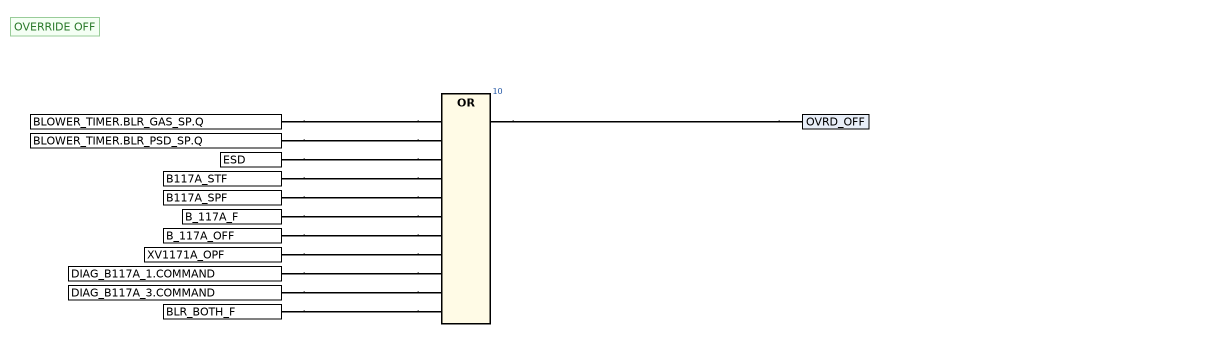
// AUTO ON
(* (BST_S_01.COMMAND OR BST_P_01.COMMAND) AND B117A_SEL OR (BST_S_01.COMPLETE OR BST_P_01.COMPLETE) AND B117A_SEL AND (B117B_STF OR XV1171B_OPF OR B_117B_OFF OR B_117B_F); result not used *)
// AUTO OFF
(* (BSP_S_10.COMMAND OR BSP_P_10.COMMAND) AND XV1171A_CLD; result not used *)
// OVERRIDE ON
(* BLOWER_TIMER.BLR_GAS_SET.Q1 AND B117A_SEL OR DIAG_B117A_2.COMMAND; result not used *)
// OVERRIDE OFF
(* BLOWER_TIMER.BLR_GAS_SP.Q OR BLOWER_TIMER.BLR_PSD_SP.Q OR ESD OR B117A_STF OR B117A_SPF OR B_117A_F OR B_117A_OFF OR XV1171A_OPF OR DIAG_B117A_1.COMMAND OR DIAG_B117A_3.COMMAND OR BLR_BOTH_F; result not used *)
B117A(
    FULL_AUTO := FULL_AUTO,
    SET_AUTO := MP_B117A_A,
    SET_MANUAL := MP_B117A_M,
    AUTO_ON := _w1,
    MANUAL_ON := MP_B117A_ST,
    INHIBIT_ON := MAINTENANCE,
    OVERRIDE_ON := _w2,
    AUTO_OFF := _w3,
    MANUAL_OFF := MP_B117A_SP,
    INHIBIT_OFF := MAINTENANCE,
    OVERRIDE_OFF := _w4,
    FEEDBACK_ON := B_117A_RUN,
    FEEDBACK_OFF := NOT B_117A_RUN); // BWTS.DEVICE
B_117A_ST := B117A.COMMAND_ON;
B117A_A := B117A.AUTO_MODE;
B117A_M := B117A.MANUAL_MODE;
B117A_RUN := B117A.INDICATOR_ON;
B117A_SPD := B117A.INDICATOR_OFF;

END_PROGRAM

// Device/Application/Logic/0.ETC/BLOWER_TIMER
PROGRAM BLOWER_TIMER
VAR
	BLR_GAS_SP: TON;
	BLR_GAS_SET: RS;		// GAS OPERATING ON
	SR_0: SR;
	BLR_PSD_SP: TON;
END_VAR
VAR // added by the converter: edge detectors and wires of the graphical bodies
    _w1 : BOOL;
END_VAR

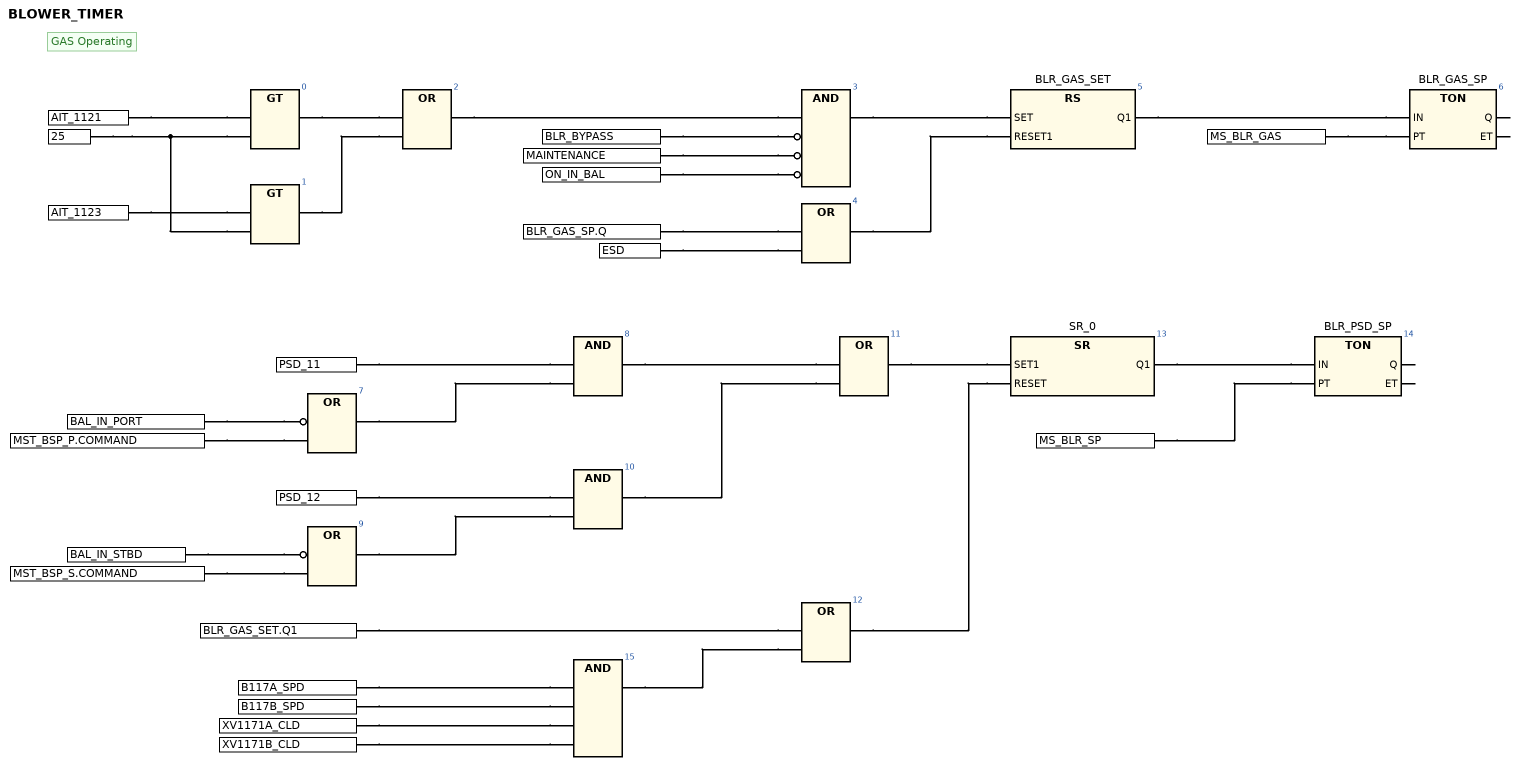
// GAS Operating
BLR_GAS_SET(SET := (AIT_1121 > 25 OR AIT_1123 > 25) AND NOT BLR_BYPASS AND NOT MAINTENANCE AND NOT ON_IN_BAL, RESET1 := BLR_GAS_SP.Q OR ESD); // RS
BLR_GAS_SP(IN := BLR_GAS_SET.Q1, PT := MS_BLR_GAS); // TON
SR_0(SET1 := PSD_11 AND (NOT BAL_IN_PORT OR MST_BSP_P.COMMAND) OR PSD_12 AND (NOT BAL_IN_STBD OR MST_BSP_S.COMMAND), RESET := BLR_GAS_SET.Q1 OR _w1); // SR
BLR_PSD_SP(IN := SR_0.Q1, PT := MS_BLR_SP); // TON
_w1 := B117A_SPD AND B117B_SPD AND XV1171A_CLD AND XV1171B_CLD;

END_PROGRAM

// Device/Application/Logic/4.Device/DEVICE_B117B
PROGRAM DEVICE_B117B
VAR
	B117B : BWTS.DEVICE;
END_VAR
VAR // added by the converter: edge detectors and wires of the graphical bodies
    _w1, _w2, _w3, _w4 : ANY;
END_VAR

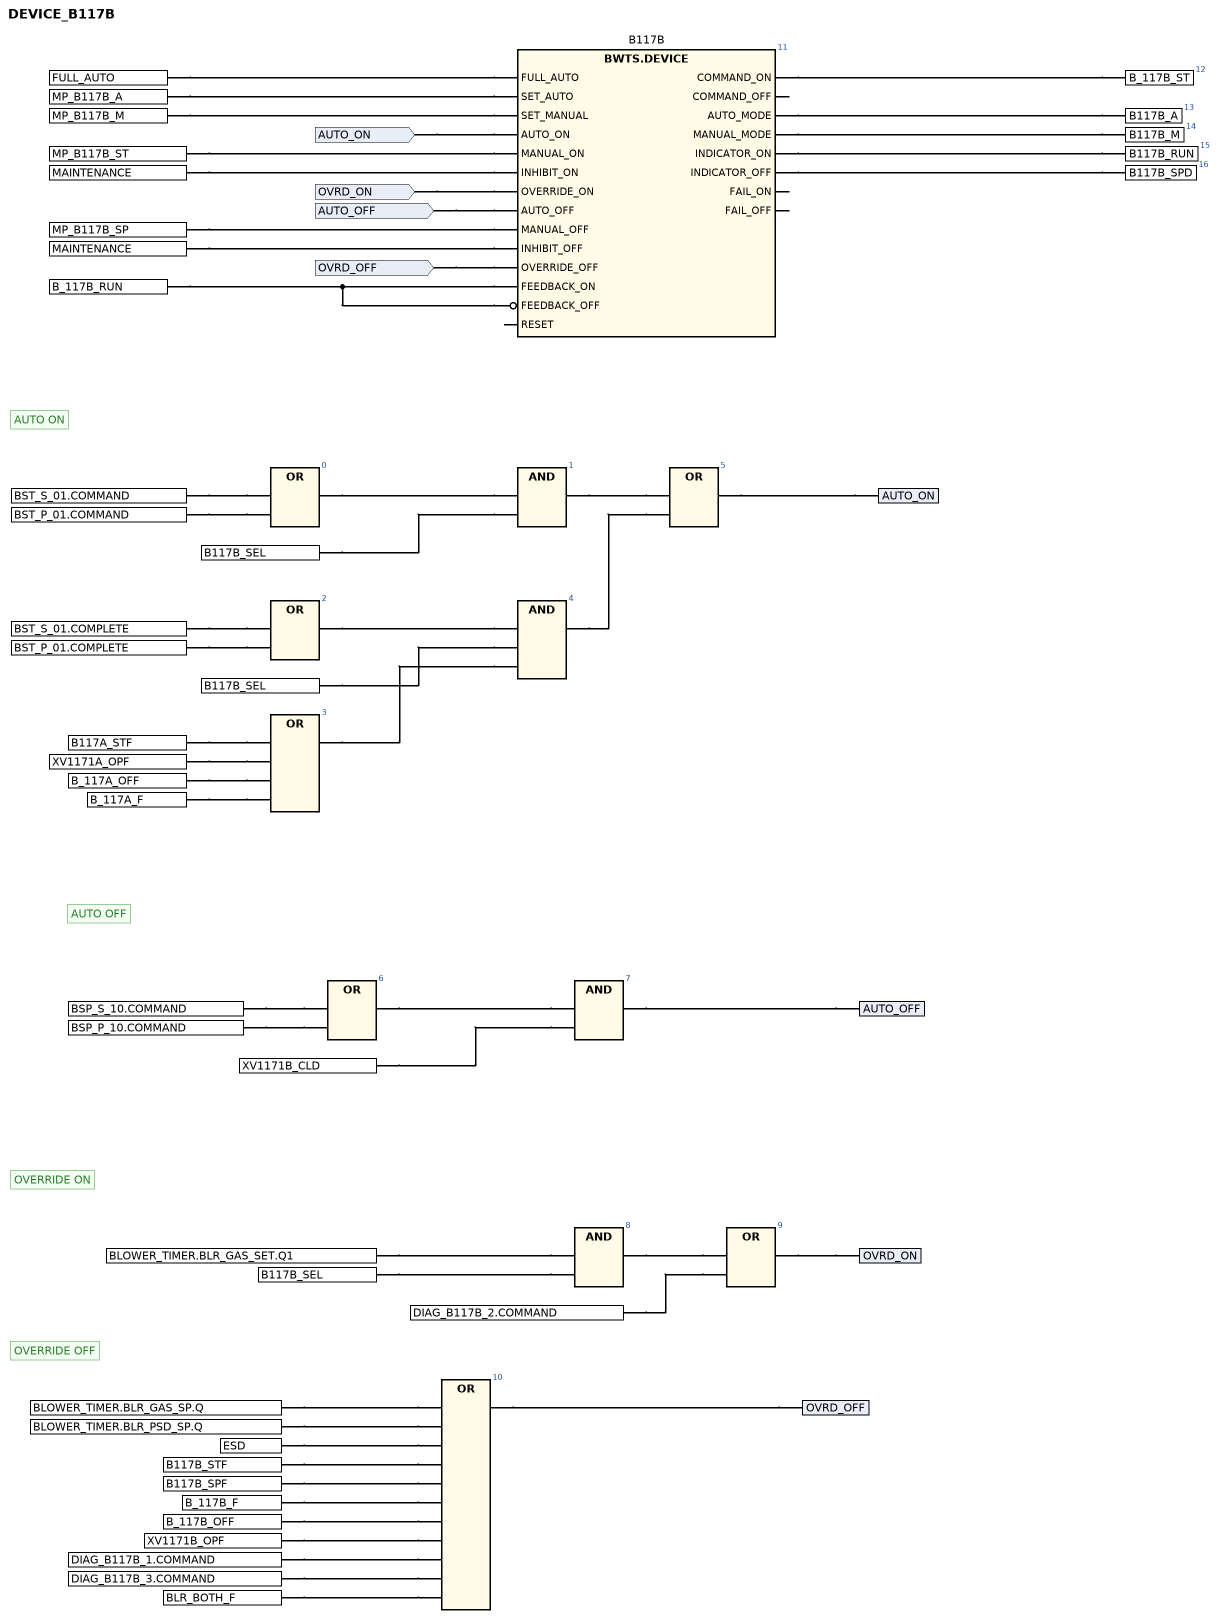
// AUTO ON
(* (BST_S_01.COMMAND OR BST_P_01.COMMAND) AND B117B_SEL OR (BST_S_01.COMPLETE OR BST_P_01.COMPLETE) AND B117B_SEL AND (B117A_STF OR XV1171A_OPF OR B_117A_OFF OR B_117A_F); result not used *)
// AUTO OFF
(* (BSP_S_10.COMMAND OR BSP_P_10.COMMAND) AND XV1171B_CLD; result not used *)
// OVERRIDE ON
(* BLOWER_TIMER.BLR_GAS_SET.Q1 AND B117B_SEL OR DIAG_B117B_2.COMMAND; result not used *)
// OVERRIDE OFF
(* BLOWER_TIMER.BLR_GAS_SP.Q OR BLOWER_TIMER.BLR_PSD_SP.Q OR ESD OR B117B_STF OR B117B_SPF OR B_117B_F OR B_117B_OFF OR XV1171B_OPF OR DIAG_B117B_1.COMMAND OR DIAG_B117B_3.COMMAND OR BLR_BOTH_F; result not used *)
B117B(
    FULL_AUTO := FULL_AUTO,
    SET_AUTO := MP_B117B_A,
    SET_MANUAL := MP_B117B_M,
    AUTO_ON := _w1,
    MANUAL_ON := MP_B117B_ST,
    INHIBIT_ON := MAINTENANCE,
    OVERRIDE_ON := _w2,
    AUTO_OFF := _w3,
    MANUAL_OFF := MP_B117B_SP,
    INHIBIT_OFF := MAINTENANCE,
    OVERRIDE_OFF := _w4,
    FEEDBACK_ON := B_117B_RUN,
    FEEDBACK_OFF := NOT B_117B_RUN); // BWTS.DEVICE
B_117B_ST := B117B.COMMAND_ON;
B117B_A := B117B.AUTO_MODE;
B117B_M := B117B.MANUAL_MODE;
B117B_RUN := B117B.INDICATOR_ON;
B117B_SPD := B117B.INDICATOR_OFF;

END_PROGRAM

// Device/Application/Logic/4.Device/DEVICE_P171A
PROGRAM DEVICE_P171A
VAR
	P171A: BWTS.DEVICE;	
	TON_0: TON;
END_VAR
VAR // added by the converter: edge detectors and wires of the graphical bodies
    _w1, _w2, _w3, _w4, _w5 : BOOL;
    _w6, _w7, _w8, _w9 : ANY;
END_VAR

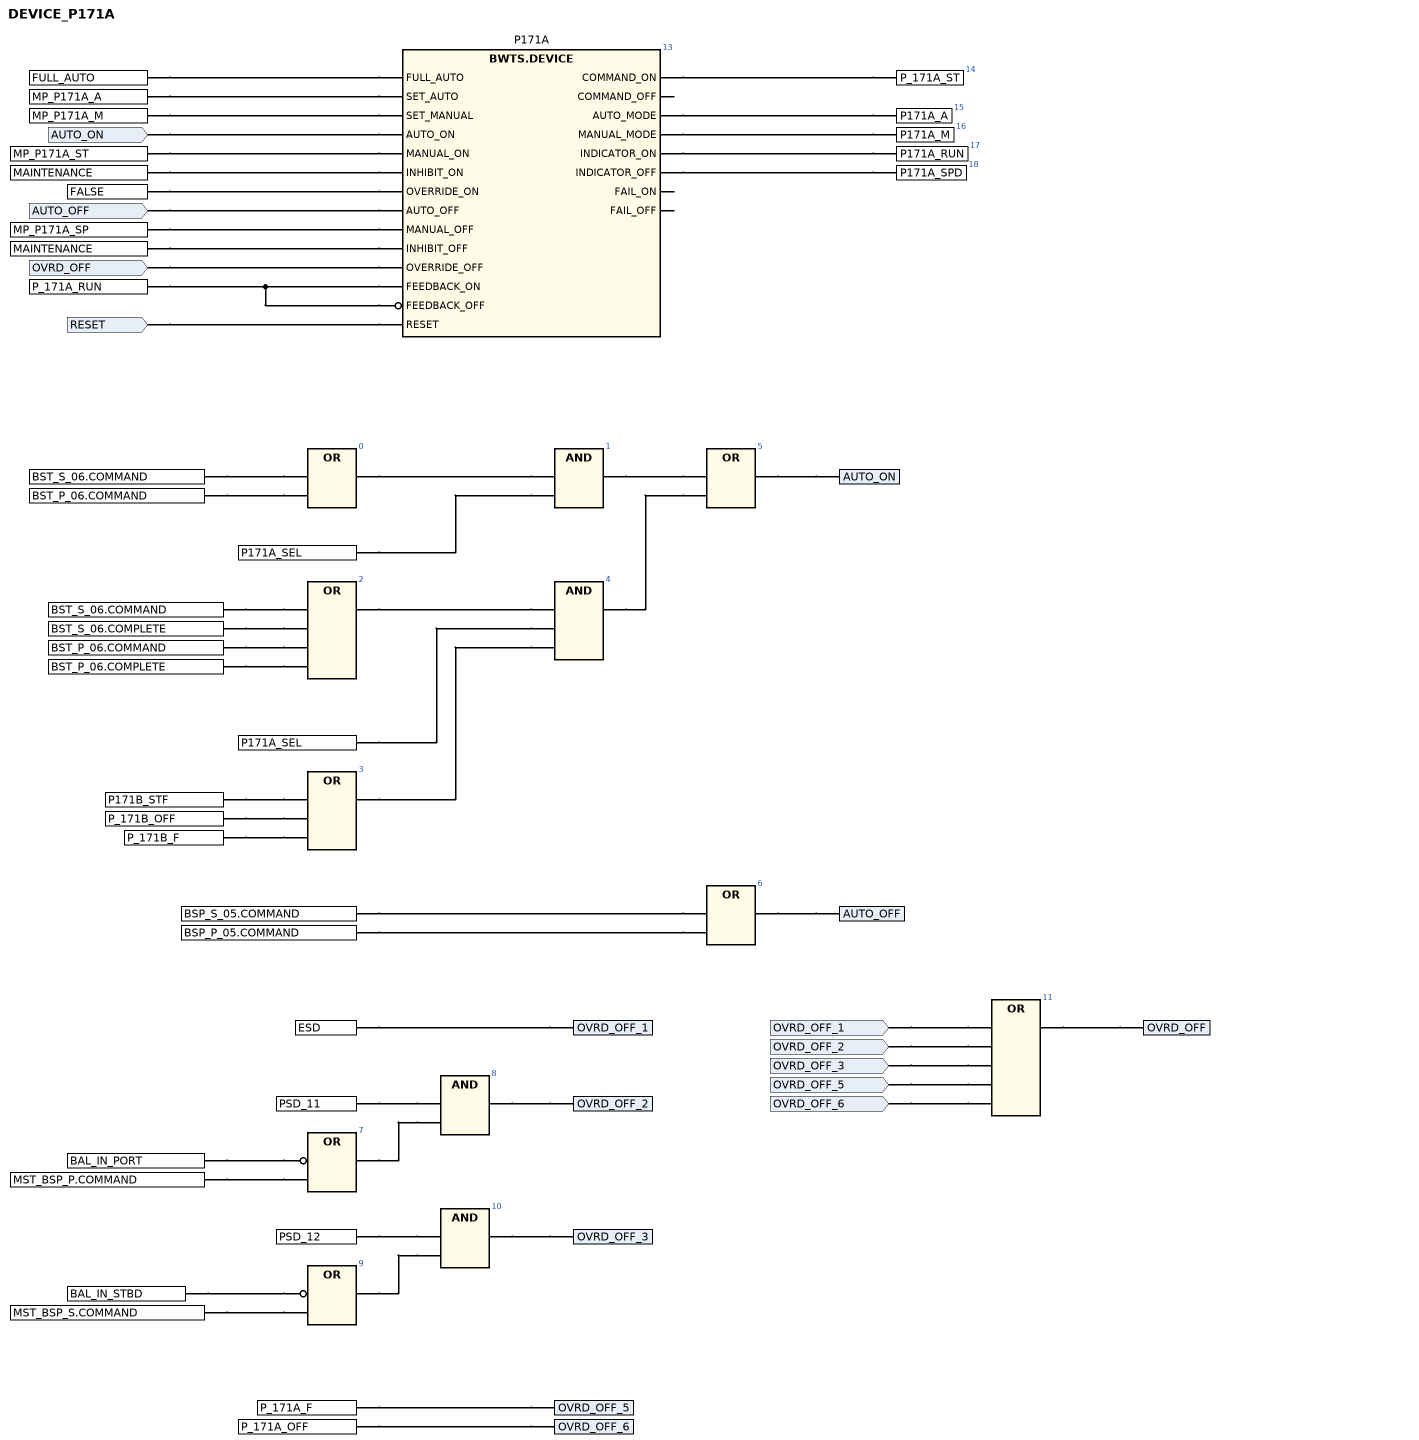
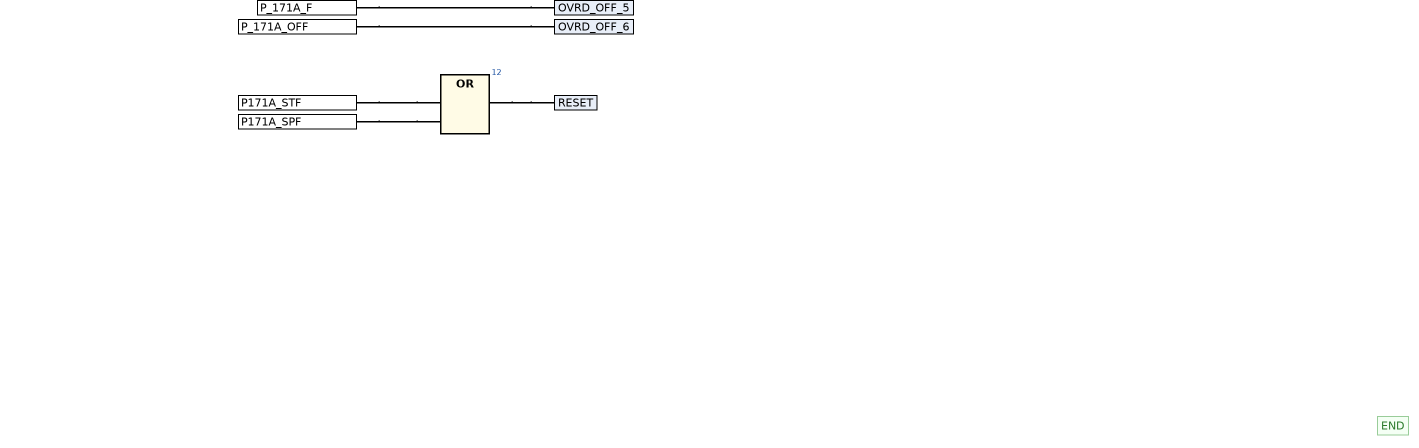
(* (BST_S_06.COMMAND OR BST_P_06.COMMAND) AND P171A_SEL OR (BST_S_06.COMMAND OR BST_S_06.COMPLETE OR BST_P_06.COMMAND OR BST_P_06.COMPLETE) AND P171A_SEL AND (P171B_STF OR P_171B_OFF OR P_171B_F); result not used *)
(* BSP_S_05.COMMAND OR BSP_P_05.COMMAND; result not used *)
(* PSD_11 AND (NOT BAL_IN_PORT OR MST_BSP_P.COMMAND); result not used *)
(* PSD_12 AND (NOT BAL_IN_STBD OR MST_BSP_S.COMMAND); result not used *)
(* _w1 OR _w2 OR _w3 OR _w4 OR _w5; result not used *)
// END
(* P171A_STF OR P171A_SPF; result not used *)
P171A(
    FULL_AUTO := FULL_AUTO,
    SET_AUTO := MP_P171A_A,
    SET_MANUAL := MP_P171A_M,
    AUTO_ON := _w6,
    MANUAL_ON := MP_P171A_ST,
    INHIBIT_ON := MAINTENANCE,
    OVERRIDE_ON := FALSE,
    AUTO_OFF := _w7,
    MANUAL_OFF := MP_P171A_SP,
    INHIBIT_OFF := MAINTENANCE,
    OVERRIDE_OFF := _w8,
    FEEDBACK_ON := P_171A_RUN,
    FEEDBACK_OFF := NOT P_171A_RUN,
    RESET := _w9); // BWTS.DEVICE
P_171A_ST := P171A.COMMAND_ON;
P171A_A := P171A.AUTO_MODE;
P171A_M := P171A.MANUAL_MODE;
P171A_RUN := P171A.INDICATOR_ON;
P171A_SPD := P171A.INDICATOR_OFF;

END_PROGRAM

// Device/Application/Logic/4.Device/DEVICE_P171B
PROGRAM DEVICE_P171B
VAR
	P171B : BWTS.DEVICE;
	AUTO_ON : BOOL;
	AUTO_OFF : BOOL;
	OVRD_OFF : BOOL;
	
	
END_VAR
VAR // added by the converter: edge detectors and wires of the graphical bodies
    _w1, _w2, _w3, _w4, _w5 : BOOL;
    _w6, _w7, _w8, _w9 : ANY;
END_VAR

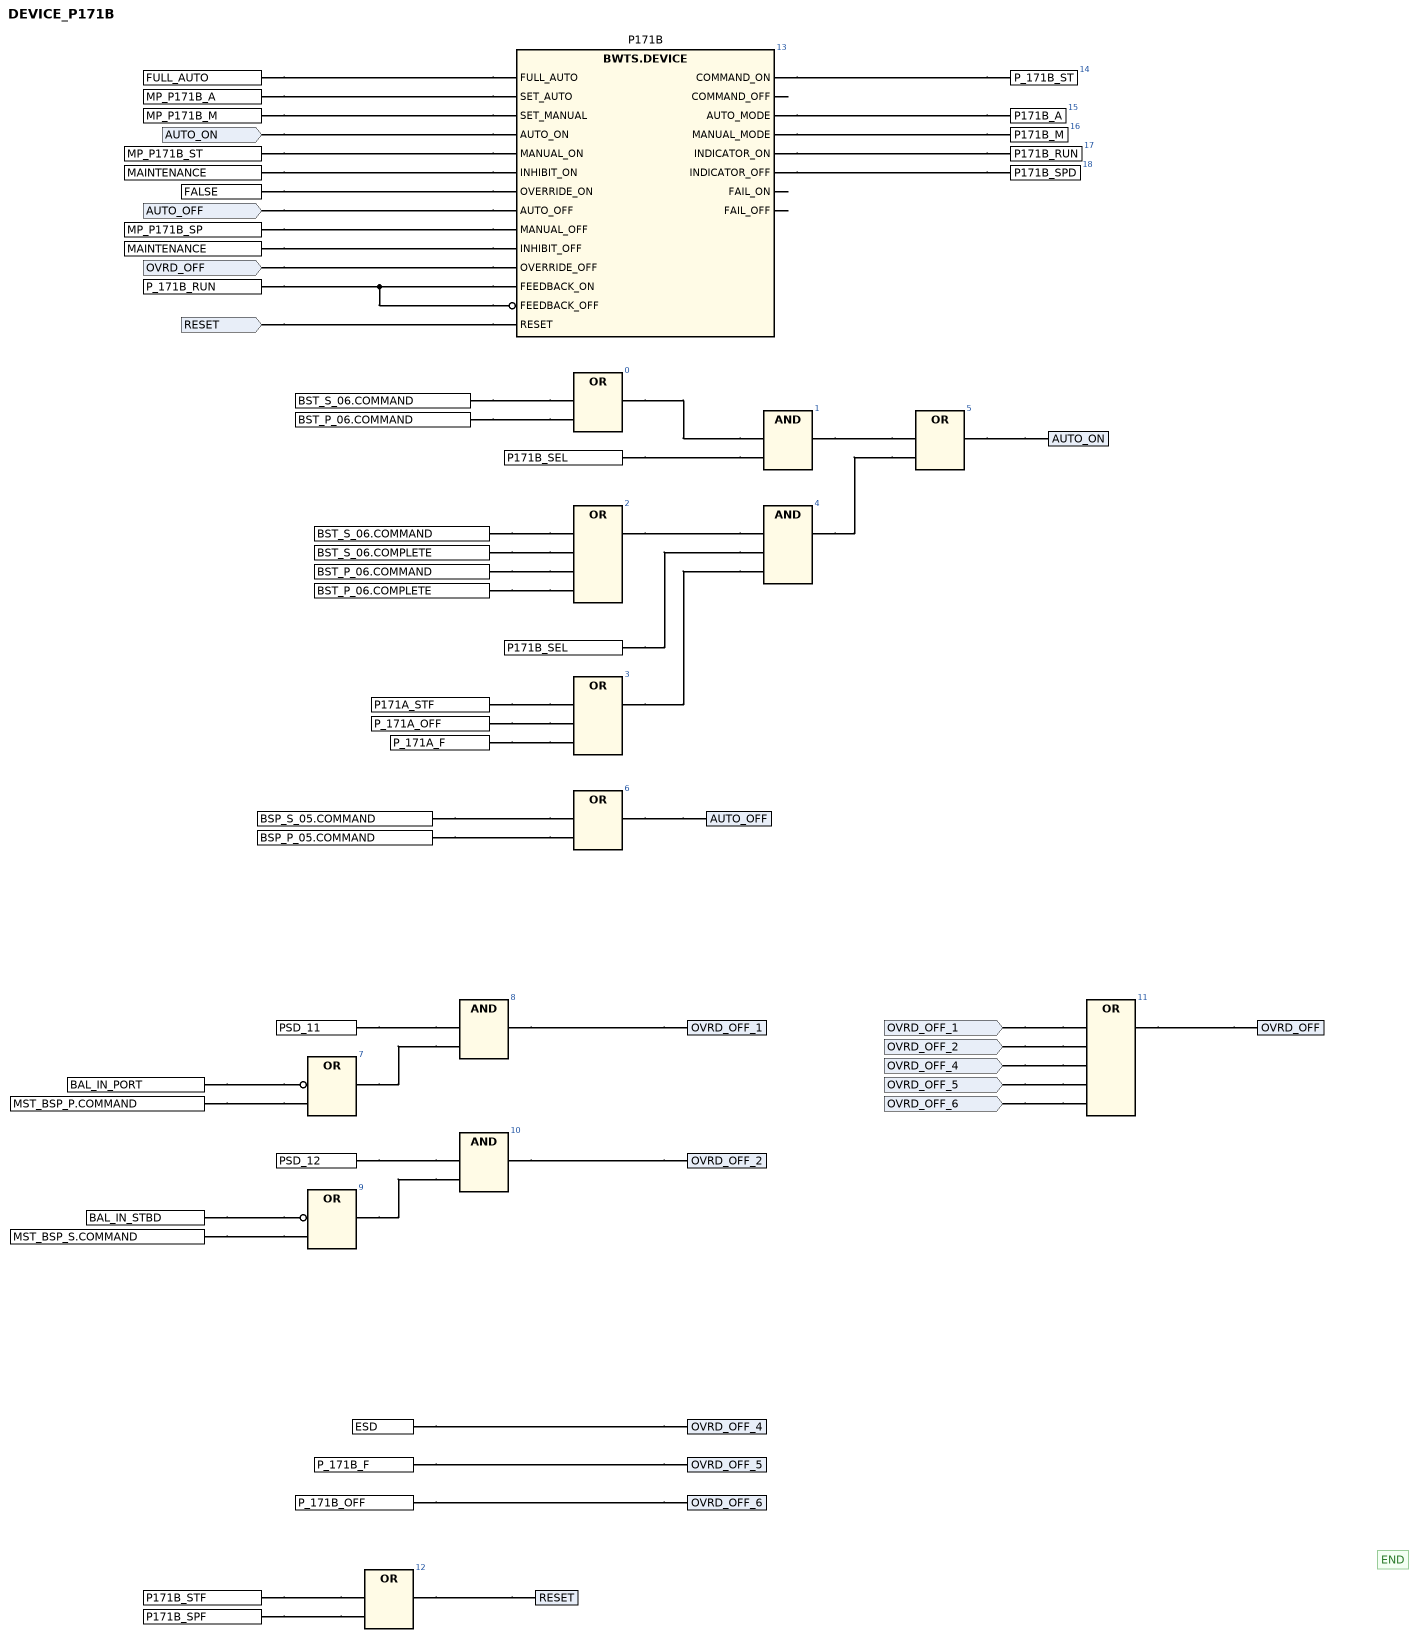
(* (BST_S_06.COMMAND OR BST_P_06.COMMAND) AND P171B_SEL OR (BST_S_06.COMMAND OR BST_S_06.COMPLETE OR BST_P_06.COMMAND OR BST_P_06.COMPLETE) AND P171B_SEL AND (P171A_STF OR P_171A_OFF OR P_171A_F); result not used *)
(* BSP_S_05.COMMAND OR BSP_P_05.COMMAND; result not used *)
(* PSD_11 AND (NOT BAL_IN_PORT OR MST_BSP_P.COMMAND); result not used *)
(* PSD_12 AND (NOT BAL_IN_STBD OR MST_BSP_S.COMMAND); result not used *)
(* _w1 OR _w2 OR _w3 OR _w4 OR _w5; result not used *)
// END
(* P171B_STF OR P171B_SPF; result not used *)
P171B(
    FULL_AUTO := FULL_AUTO,
    SET_AUTO := MP_P171B_A,
    SET_MANUAL := MP_P171B_M,
    AUTO_ON := _w6,
    MANUAL_ON := MP_P171B_ST,
    INHIBIT_ON := MAINTENANCE,
    OVERRIDE_ON := FALSE,
    AUTO_OFF := _w7,
    MANUAL_OFF := MP_P171B_SP,
    INHIBIT_OFF := MAINTENANCE,
    OVERRIDE_OFF := _w8,
    FEEDBACK_ON := P_171B_RUN,
    FEEDBACK_OFF := NOT P_171B_RUN,
    RESET := _w9); // BWTS.DEVICE
P_171B_ST := P171B.COMMAND_ON;
P171B_A := P171B.AUTO_MODE;
P171B_M := P171B.MANUAL_MODE;
P171B_RUN := P171B.INDICATOR_ON;
P171B_SPD := P171B.INDICATOR_OFF;

END_PROGRAM

// Device/Application/Logic/4.Device/DEVICE_RFA
PROGRAM DEVICE_RFA
VAR
	RF142A: BWTS.DEVICE;
	RFA_CONT: BWTS.RF_CONT;
	TON_0: TON;
END_VAR
VAR // added by the converter: edge detectors and wires of the graphical bodies
    _w1, _w7, _w8, _w9, _w10, _w11, _w12, _w13, _w14, _w15, _w16 : ANY;
    _w2, _w3, _w4, _w5, _w6 : BOOL;
END_VAR

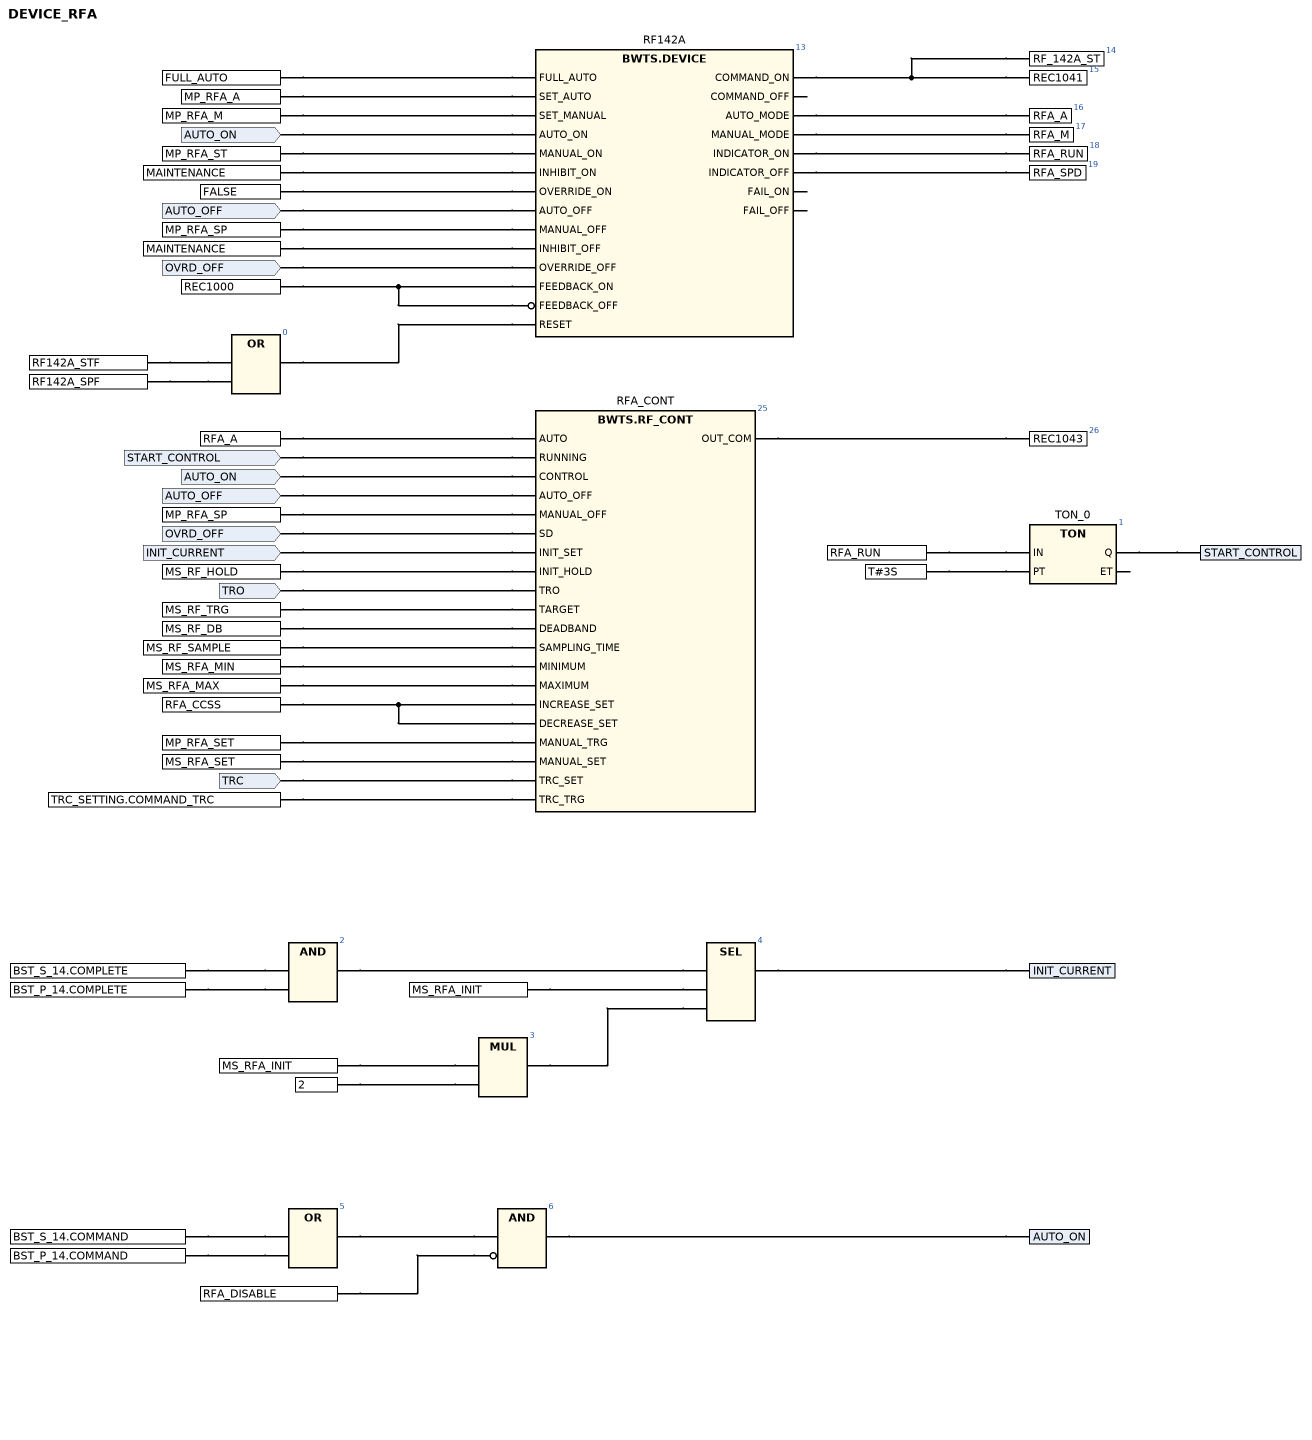
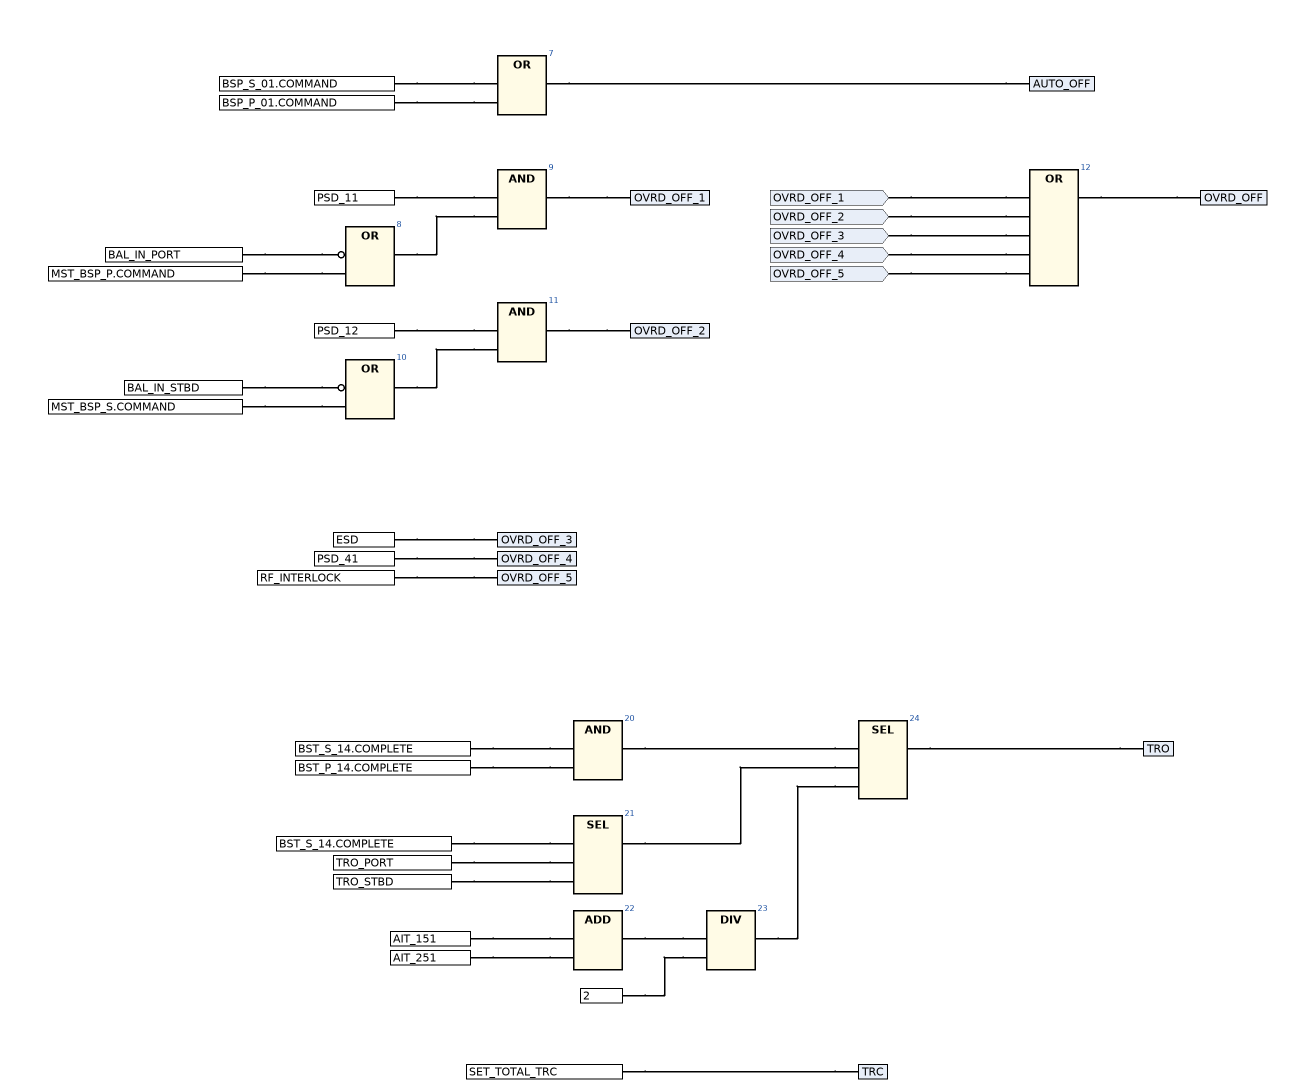
_w1 := RF142A_STF OR RF142A_SPF;
TON_0(IN := RFA_RUN, PT := T#3S); // TON
(* SEL(BST_S_14.COMPLETE AND BST_P_14.COMPLETE, MS_RFA_INIT, MS_RFA_INIT * 2); result not used *)
(* (BST_S_14.COMMAND OR BST_P_14.COMMAND) AND NOT RFA_DISABLE; result not used *)
(* BSP_S_01.COMMAND OR BSP_P_01.COMMAND; result not used *)
(* PSD_11 AND (NOT BAL_IN_PORT OR MST_BSP_P.COMMAND); result not used *)
(* PSD_12 AND (NOT BAL_IN_STBD OR MST_BSP_S.COMMAND); result not used *)
(* _w2 OR _w3 OR _w4 OR _w5 OR _w6; result not used *)
RF142A(
    FULL_AUTO := FULL_AUTO,
    SET_AUTO := MP_RFA_A,
    SET_MANUAL := MP_RFA_M,
    AUTO_ON := _w7,
    MANUAL_ON := MP_RFA_ST,
    INHIBIT_ON := MAINTENANCE,
    OVERRIDE_ON := FALSE,
    AUTO_OFF := _w8,
    MANUAL_OFF := MP_RFA_SP,
    INHIBIT_OFF := MAINTENANCE,
    OVERRIDE_OFF := _w9,
    FEEDBACK_ON := REC1000,
    FEEDBACK_OFF := NOT REC1000,
    RESET := _w1); // BWTS.DEVICE
RF_142A_ST := RF142A.COMMAND_ON;
REC1041 := RF142A.COMMAND_ON;
RFA_A := RF142A.AUTO_MODE;
RFA_M := RF142A.MANUAL_MODE;
RFA_RUN := RF142A.INDICATOR_ON;
RFA_SPD := RF142A.INDICATOR_OFF;
(* SEL(BST_S_14.COMPLETE AND BST_P_14.COMPLETE, SEL(BST_S_14.COMPLETE, TRO_PORT, TRO_STBD), (AIT_151 + AIT_251) / 2); result not used *)
RFA_CONT(
    AUTO := RFA_A,
    RUNNING := _w10,
    CONTROL := _w11,
    AUTO_OFF := _w12,
    MANUAL_OFF := MP_RFA_SP,
    SD := _w13,
    INIT_SET := _w14,
    INIT_HOLD := MS_RF_HOLD,
    TRO := _w15,
    TARGET := MS_RF_TRG,
    DEADBAND := MS_RF_DB,
    SAMPLING_TIME := MS_RF_SAMPLE,
    MINIMUM := MS_RFA_MIN,
    MAXIMUM := MS_RFA_MAX,
    INCREASE_SET := RFA_CCSS,
    DECREASE_SET := RFA_CCSS,
    MANUAL_TRG := MP_RFA_SET,
    MANUAL_SET := MS_RFA_SET,
    TRC_SET := _w16,
    TRC_TRG := TRC_SETTING.COMMAND_TRC); // BWTS.RF_CONT
REC1043 := RFA_CONT.OUT_COM;

END_PROGRAM

// Device/Application/Logic/0.ETC/TRC_SETTING
PROGRAM TRC_SETTING
VAR
	TRC_SET_R0_0: BWTS.TRC_SET;
	ENABLE_STBD : BOOL;
	ENABLE_PORT : BOOL;
	ENABLE_APT : BOOL;
	COMMAND_TRC : BOOL;
	TP_0: TP;
	TP_1: TP;
	TP_2: TP;
	TP_3: TP;
END_VAR
VAR // added by the converter: edge detectors and wires of the graphical bodies
    _w1, _w2, _w3, _w4 : BOOL;
END_VAR

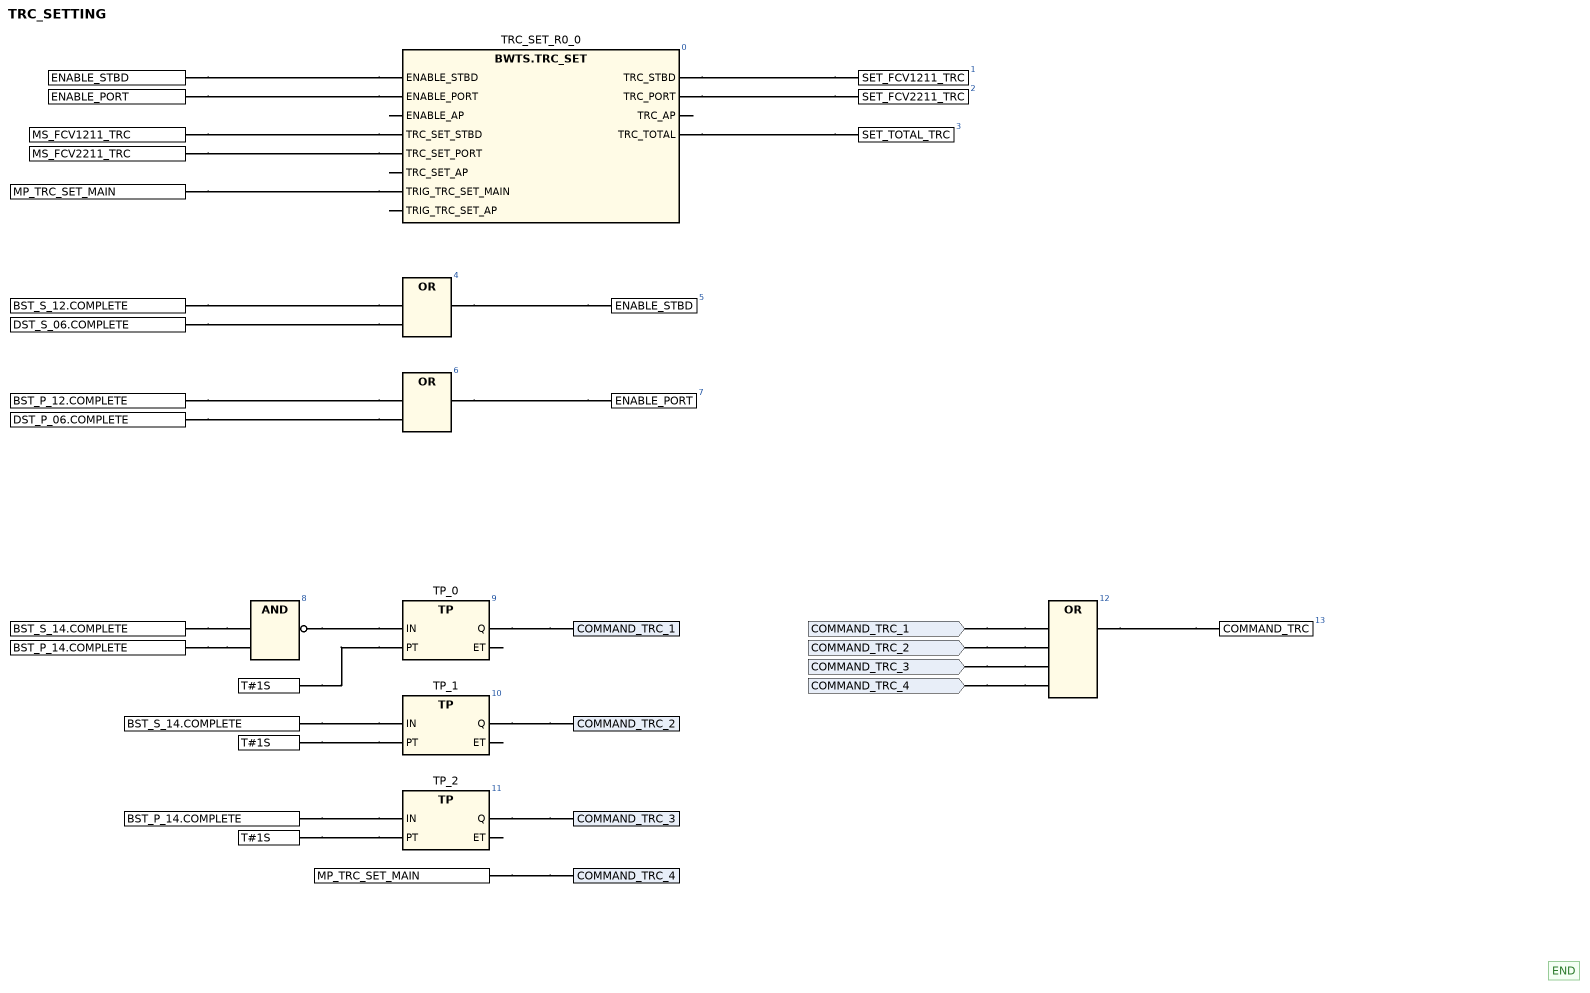
TRC_SET_R0_0(
    ENABLE_STBD := ENABLE_STBD,
    ENABLE_PORT := ENABLE_PORT,
    TRC_SET_STBD := MS_FCV1211_TRC,
    TRC_SET_PORT := MS_FCV2211_TRC,
    TRIG_TRC_SET_MAIN := MP_TRC_SET_MAIN); // BWTS.TRC_SET
SET_FCV1211_TRC := TRC_SET_R0_0.TRC_STBD;
SET_FCV2211_TRC := TRC_SET_R0_0.TRC_PORT;
SET_TOTAL_TRC := TRC_SET_R0_0.TRC_TOTAL;
ENABLE_STBD := BST_S_12.COMPLETE OR DST_S_06.COMPLETE;
ENABLE_PORT := BST_P_12.COMPLETE OR DST_P_06.COMPLETE;
TP_0(IN := NOT (BST_S_14.COMPLETE AND BST_P_14.COMPLETE), PT := T#1S); // TP
TP_1(IN := BST_S_14.COMPLETE, PT := T#1S); // TP
// END
TP_2(IN := BST_P_14.COMPLETE, PT := T#1S); // TP
COMMAND_TRC := _w1 OR _w2 OR _w3 OR _w4;

END_PROGRAM

// Device/Application/Logic/4.Device/DEVICE_RFB
PROGRAM DEVICE_RFB
VAR
	RF142B: BWTS.DEVICE;
	RFB_CONT: BWTS.RF_CONT;
	TON_0 : TON;
END_VAR
VAR // added by the converter: edge detectors and wires of the graphical bodies
    _w1, _w7, _w8, _w9, _w10, _w11, _w12, _w13, _w14, _w15, _w16 : ANY;
    _w2, _w3, _w4, _w5, _w6 : BOOL;
END_VAR

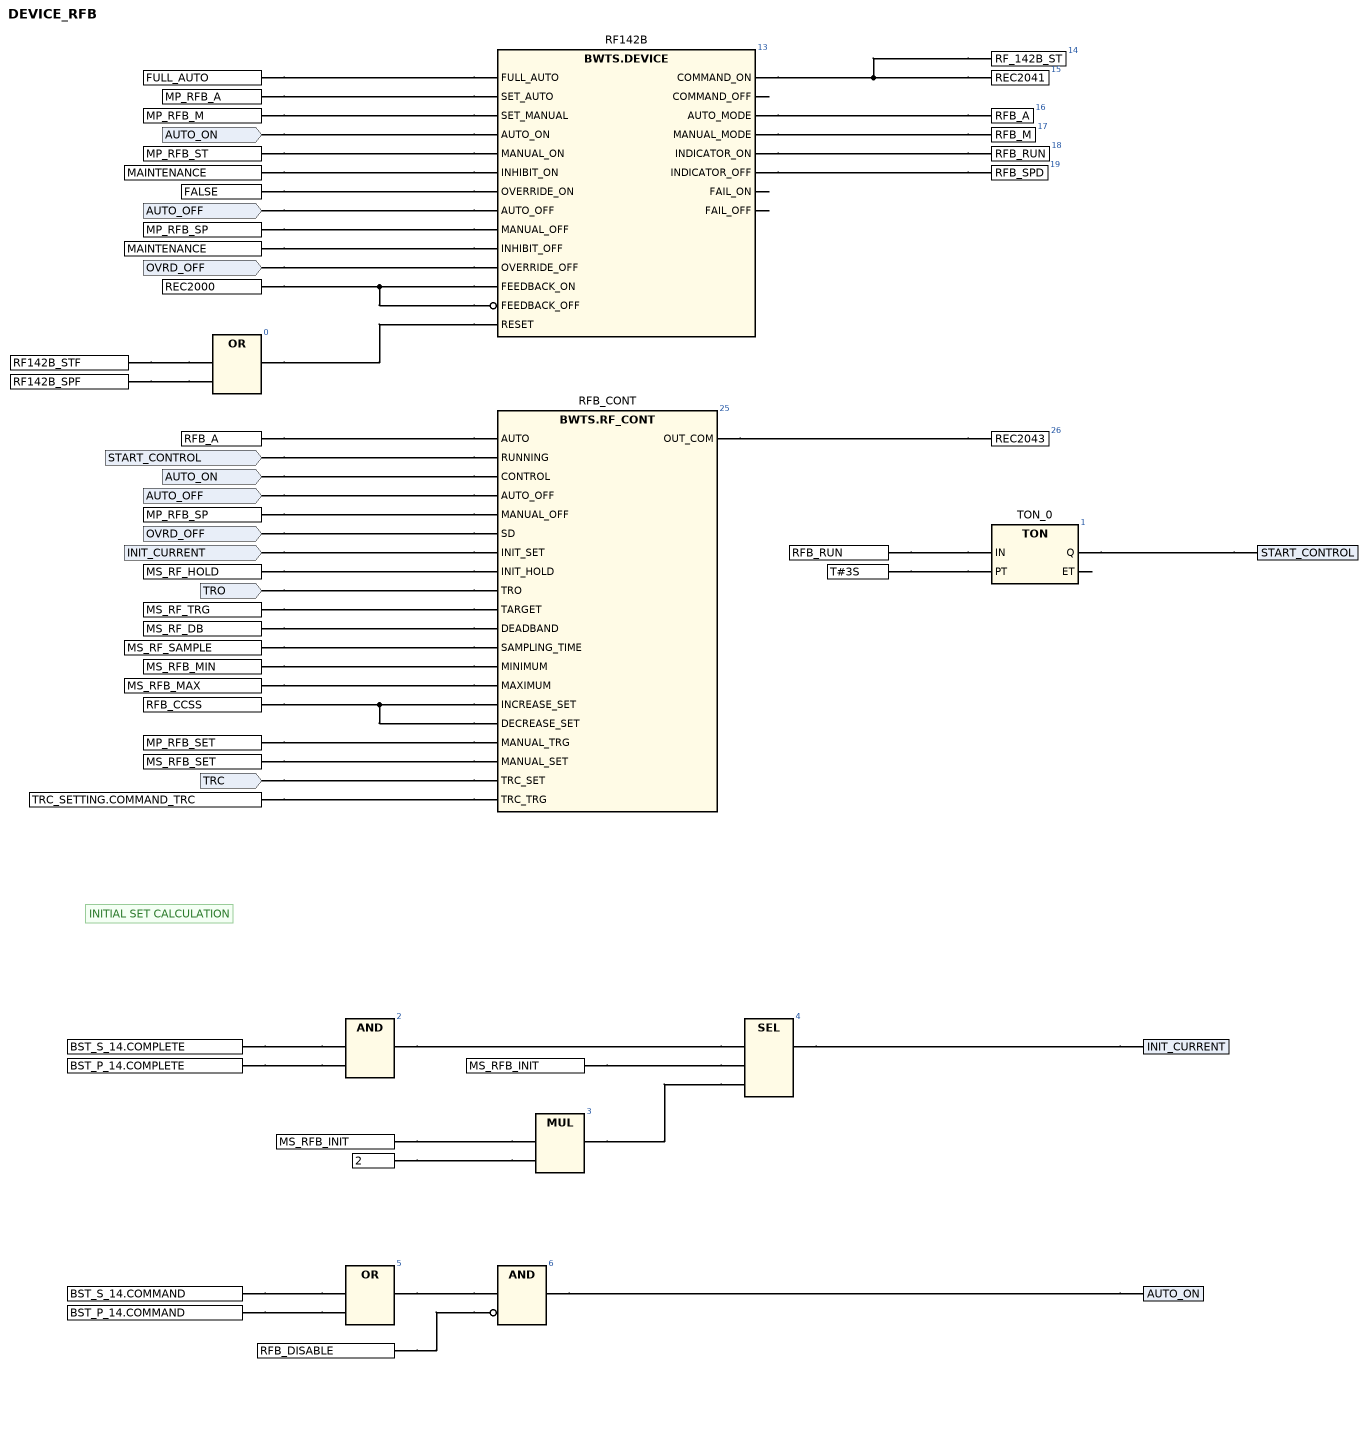
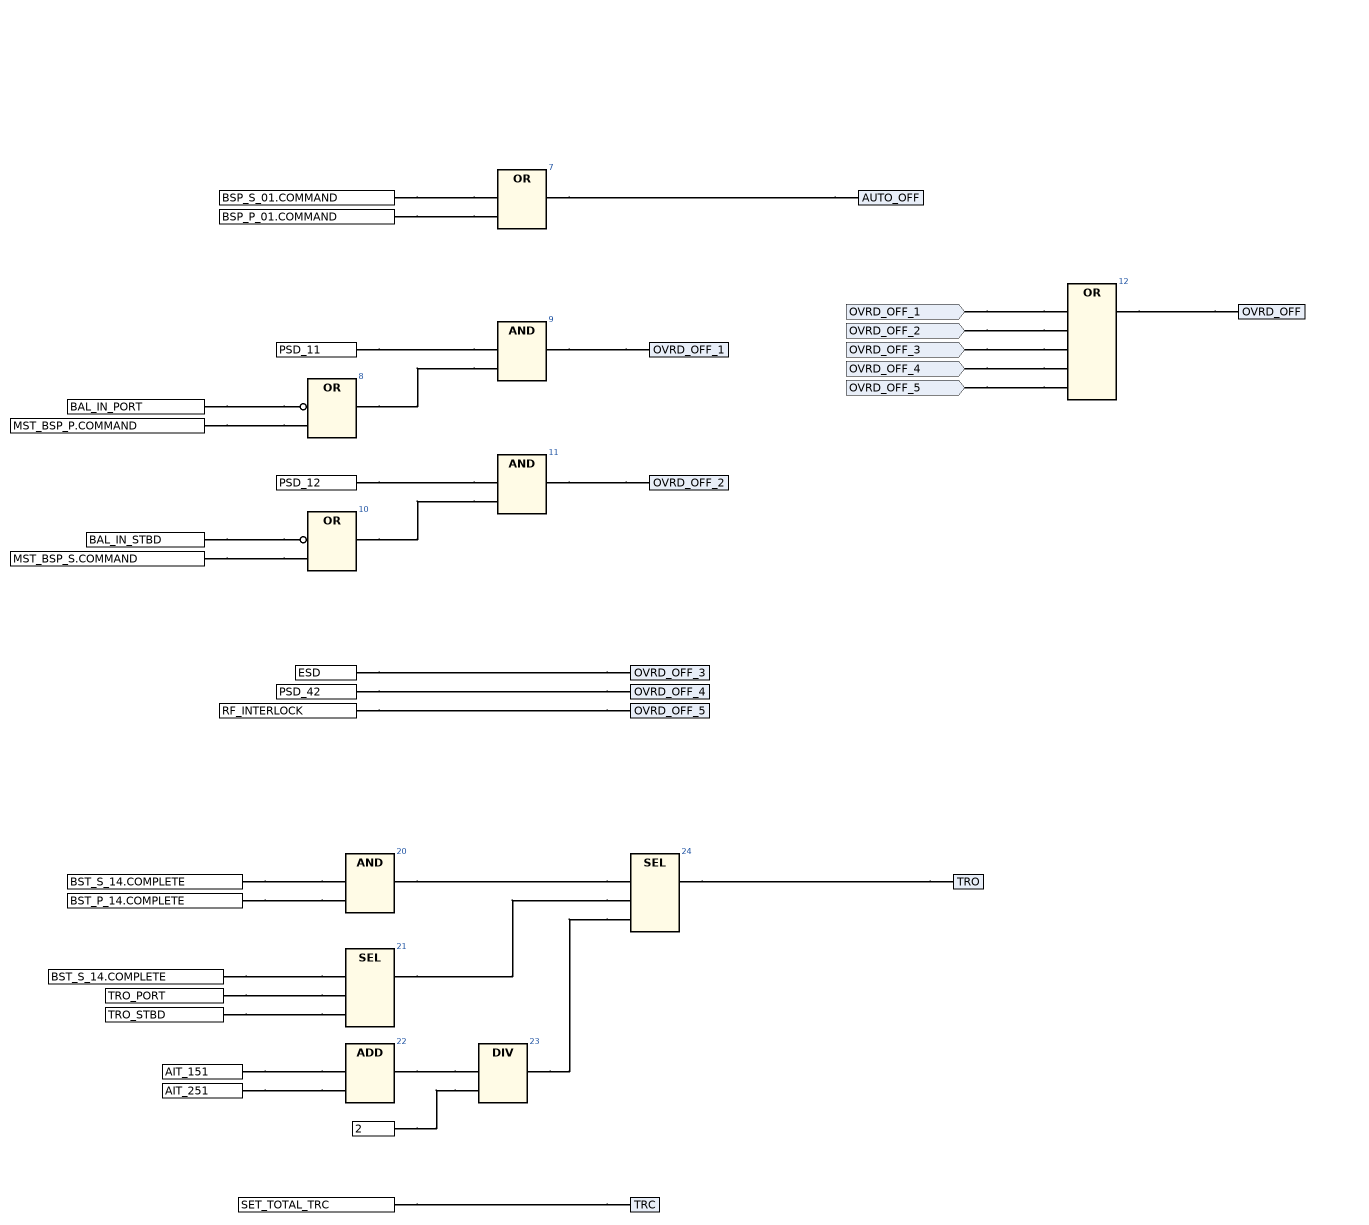
_w1 := RF142B_STF OR RF142B_SPF;
TON_0(IN := RFB_RUN, PT := T#3S); // TON
// INITIAL SET CALCULATION
(* SEL(BST_S_14.COMPLETE AND BST_P_14.COMPLETE, MS_RFB_INIT, MS_RFB_INIT * 2); result not used *)
(* (BST_S_14.COMMAND OR BST_P_14.COMMAND) AND NOT RFB_DISABLE; result not used *)
(* BSP_S_01.COMMAND OR BSP_P_01.COMMAND; result not used *)
(* PSD_11 AND (NOT BAL_IN_PORT OR MST_BSP_P.COMMAND); result not used *)
(* PSD_12 AND (NOT BAL_IN_STBD OR MST_BSP_S.COMMAND); result not used *)
(* _w2 OR _w3 OR _w4 OR _w5 OR _w6; result not used *)
RF142B(
    FULL_AUTO := FULL_AUTO,
    SET_AUTO := MP_RFB_A,
    SET_MANUAL := MP_RFB_M,
    AUTO_ON := _w7,
    MANUAL_ON := MP_RFB_ST,
    INHIBIT_ON := MAINTENANCE,
    OVERRIDE_ON := FALSE,
    AUTO_OFF := _w8,
    MANUAL_OFF := MP_RFB_SP,
    INHIBIT_OFF := MAINTENANCE,
    OVERRIDE_OFF := _w9,
    FEEDBACK_ON := REC2000,
    FEEDBACK_OFF := NOT REC2000,
    RESET := _w1); // BWTS.DEVICE
RF_142B_ST := RF142B.COMMAND_ON;
REC2041 := RF142B.COMMAND_ON;
RFB_A := RF142B.AUTO_MODE;
RFB_M := RF142B.MANUAL_MODE;
RFB_RUN := RF142B.INDICATOR_ON;
RFB_SPD := RF142B.INDICATOR_OFF;
(* SEL(BST_S_14.COMPLETE AND BST_P_14.COMPLETE, SEL(BST_S_14.COMPLETE, TRO_PORT, TRO_STBD), (AIT_151 + AIT_251) / 2); result not used *)
RFB_CONT(
    AUTO := RFB_A,
    RUNNING := _w10,
    CONTROL := _w11,
    AUTO_OFF := _w12,
    MANUAL_OFF := MP_RFB_SP,
    SD := _w13,
    INIT_SET := _w14,
    INIT_HOLD := MS_RF_HOLD,
    TRO := _w15,
    TARGET := MS_RF_TRG,
    DEADBAND := MS_RF_DB,
    SAMPLING_TIME := MS_RF_SAMPLE,
    MINIMUM := MS_RFB_MIN,
    MAXIMUM := MS_RFB_MAX,
    INCREASE_SET := RFB_CCSS,
    DECREASE_SET := RFB_CCSS,
    MANUAL_TRG := MP_RFB_SET,
    MANUAL_SET := MS_RFB_SET,
    TRC_SET := _w16,
    TRC_TRG := TRC_SETTING.COMMAND_TRC); // BWTS.RF_CONT
REC2043 := RFB_CONT.OUT_COM;

END_PROGRAM

// Device/Application/Logic/4.Device/DEVICE_RFC
PROGRAM DEVICE_RFC
VAR
	RF142C: BWTS.DEVICE;
	RFC_CONT: BWTS.RF_CONT;
	TON_0: TON;
END_VAR
VAR // added by the converter: edge detectors and wires of the graphical bodies
    _w1, _w7, _w8, _w9, _w10, _w11, _w12, _w13, _w14, _w15, _w16 : ANY;
    _w2, _w3, _w4, _w5, _w6 : BOOL;
END_VAR

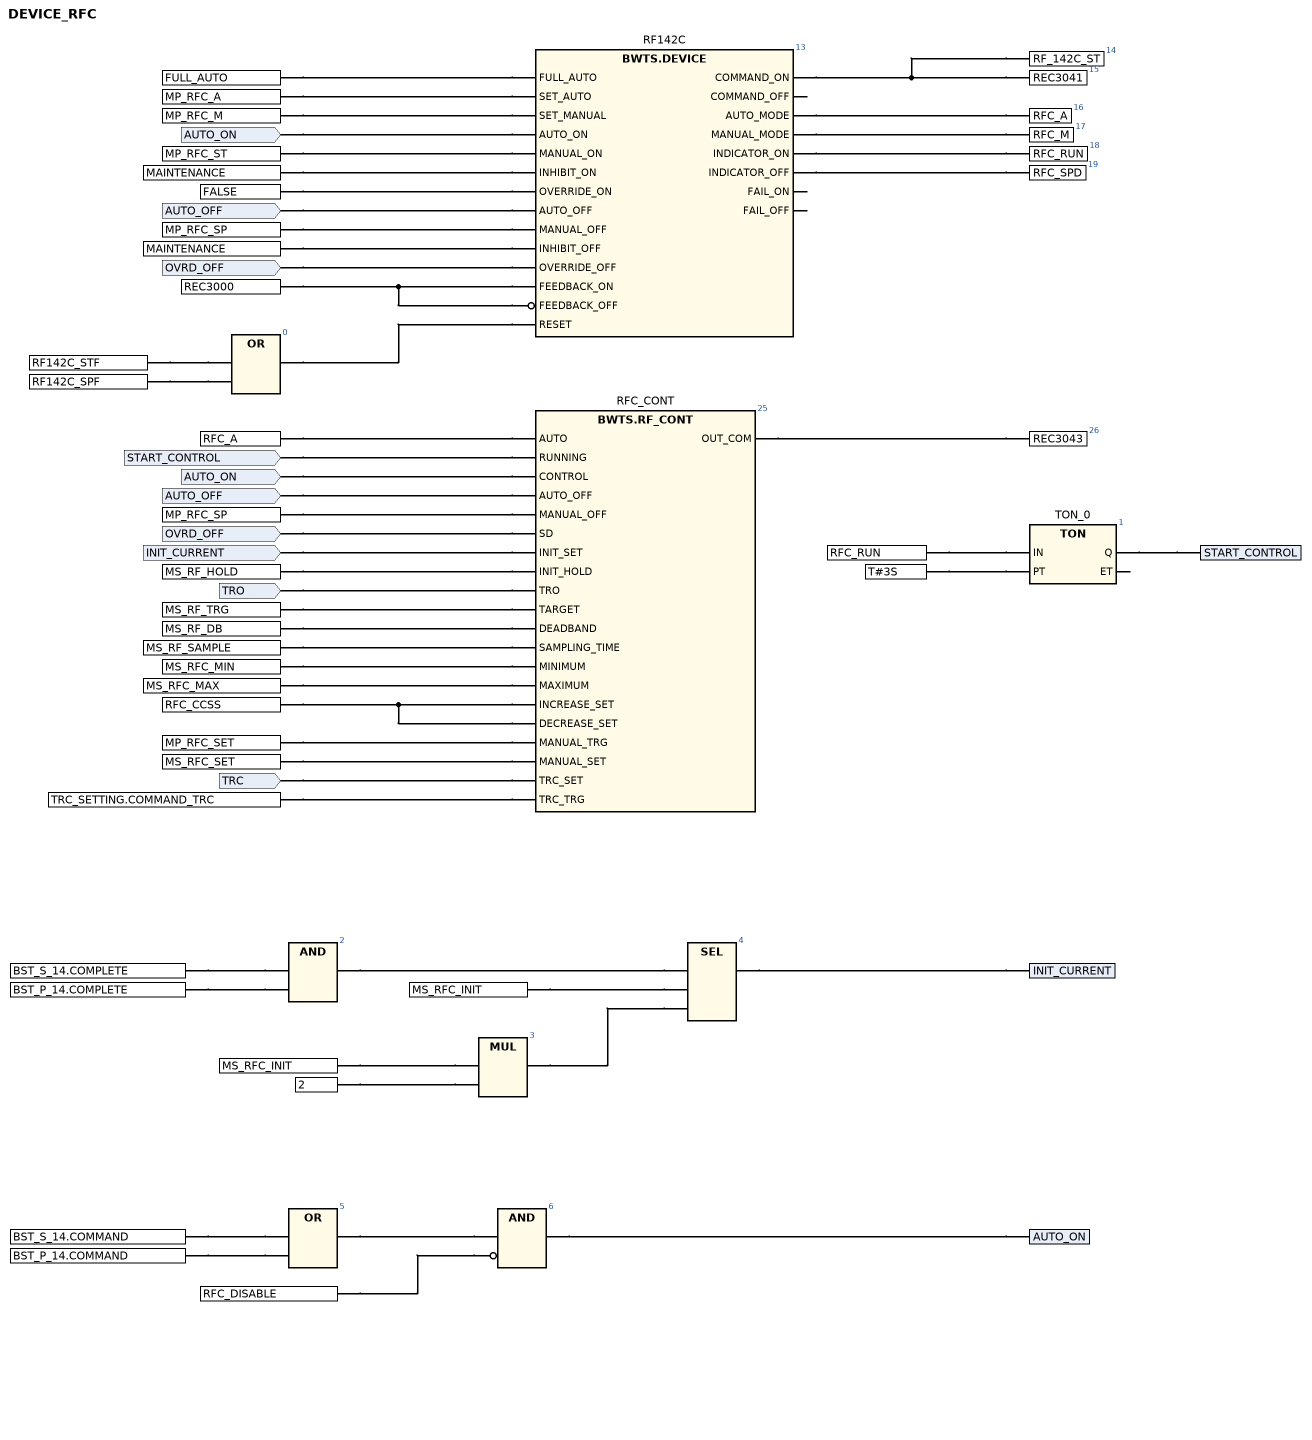
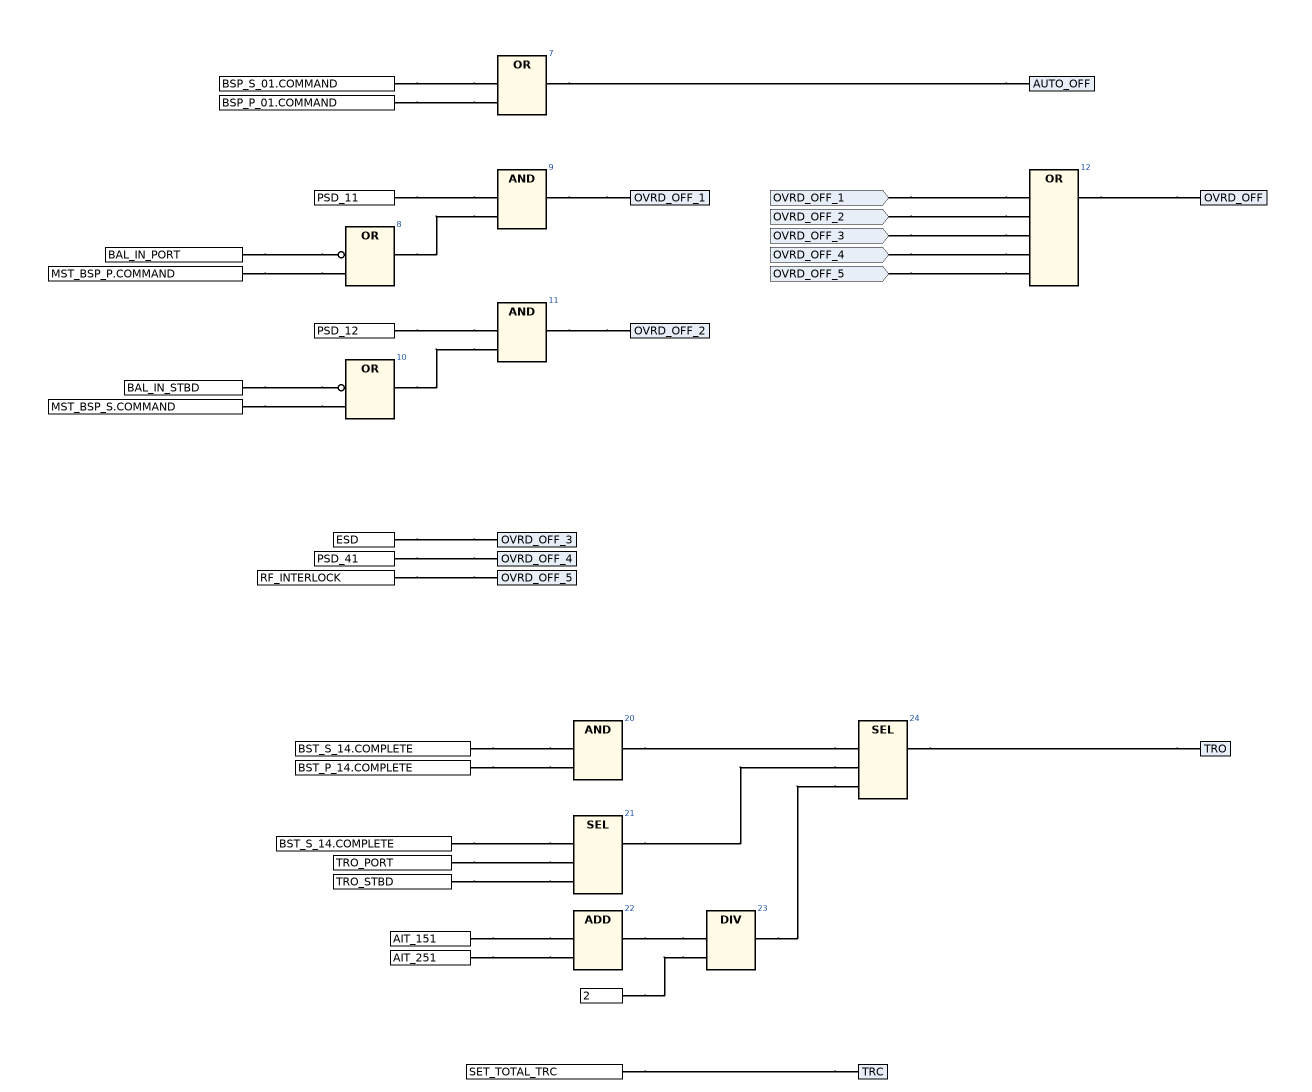
_w1 := RF142C_STF OR RF142C_SPF;
TON_0(IN := RFC_RUN, PT := T#3S); // TON
(* SEL(BST_S_14.COMPLETE AND BST_P_14.COMPLETE, MS_RFC_INIT, MS_RFC_INIT * 2); result not used *)
(* (BST_S_14.COMMAND OR BST_P_14.COMMAND) AND NOT RFC_DISABLE; result not used *)
(* BSP_S_01.COMMAND OR BSP_P_01.COMMAND; result not used *)
(* PSD_11 AND (NOT BAL_IN_PORT OR MST_BSP_P.COMMAND); result not used *)
(* PSD_12 AND (NOT BAL_IN_STBD OR MST_BSP_S.COMMAND); result not used *)
(* _w2 OR _w3 OR _w4 OR _w5 OR _w6; result not used *)
RF142C(
    FULL_AUTO := FULL_AUTO,
    SET_AUTO := MP_RFC_A,
    SET_MANUAL := MP_RFC_M,
    AUTO_ON := _w7,
    MANUAL_ON := MP_RFC_ST,
    INHIBIT_ON := MAINTENANCE,
    OVERRIDE_ON := FALSE,
    AUTO_OFF := _w8,
    MANUAL_OFF := MP_RFC_SP,
    INHIBIT_OFF := MAINTENANCE,
    OVERRIDE_OFF := _w9,
    FEEDBACK_ON := REC3000,
    FEEDBACK_OFF := NOT REC3000,
    RESET := _w1); // BWTS.DEVICE
RF_142C_ST := RF142C.COMMAND_ON;
REC3041 := RF142C.COMMAND_ON;
RFC_A := RF142C.AUTO_MODE;
RFC_M := RF142C.MANUAL_MODE;
RFC_RUN := RF142C.INDICATOR_ON;
RFC_SPD := RF142C.INDICATOR_OFF;
(* SEL(BST_S_14.COMPLETE AND BST_P_14.COMPLETE, SEL(BST_S_14.COMPLETE, TRO_PORT, TRO_STBD), (AIT_151 + AIT_251) / 2); result not used *)
RFC_CONT(
    AUTO := RFC_A,
    RUNNING := _w10,
    CONTROL := _w11,
    AUTO_OFF := _w12,
    MANUAL_OFF := MP_RFC_SP,
    SD := _w13,
    INIT_SET := _w14,
    INIT_HOLD := MS_RF_HOLD,
    TRO := _w15,
    TARGET := MS_RF_TRG,
    DEADBAND := MS_RF_DB,
    SAMPLING_TIME := MS_RF_SAMPLE,
    MINIMUM := MS_RFC_MIN,
    MAXIMUM := MS_RFC_MAX,
    INCREASE_SET := RFC_CCSS,
    DECREASE_SET := RFC_CCSS,
    MANUAL_TRG := MP_RFC_SET,
    MANUAL_SET := MS_RFC_SET,
    TRC_SET := _w16,
    TRC_TRG := TRC_SETTING.COMMAND_TRC); // BWTS.RF_CONT
REC3043 := RFC_CONT.OUT_COM;

END_PROGRAM

// Device/Application/Logic/4.Device/DEVICE_P132
PROGRAM DEVICE_P132
VAR
	P132: BWTS.DEVICE;
	STEP_NU_R0_0: BWTS.STEP_NU;
END_VAR
VAR // added by the converter: edge detectors and wires of the graphical bodies
    _w1, _w2, _w3, _w4, _w5, _w6, _w7, _w8, _w9, _w10, _w11 : ANY;
END_VAR

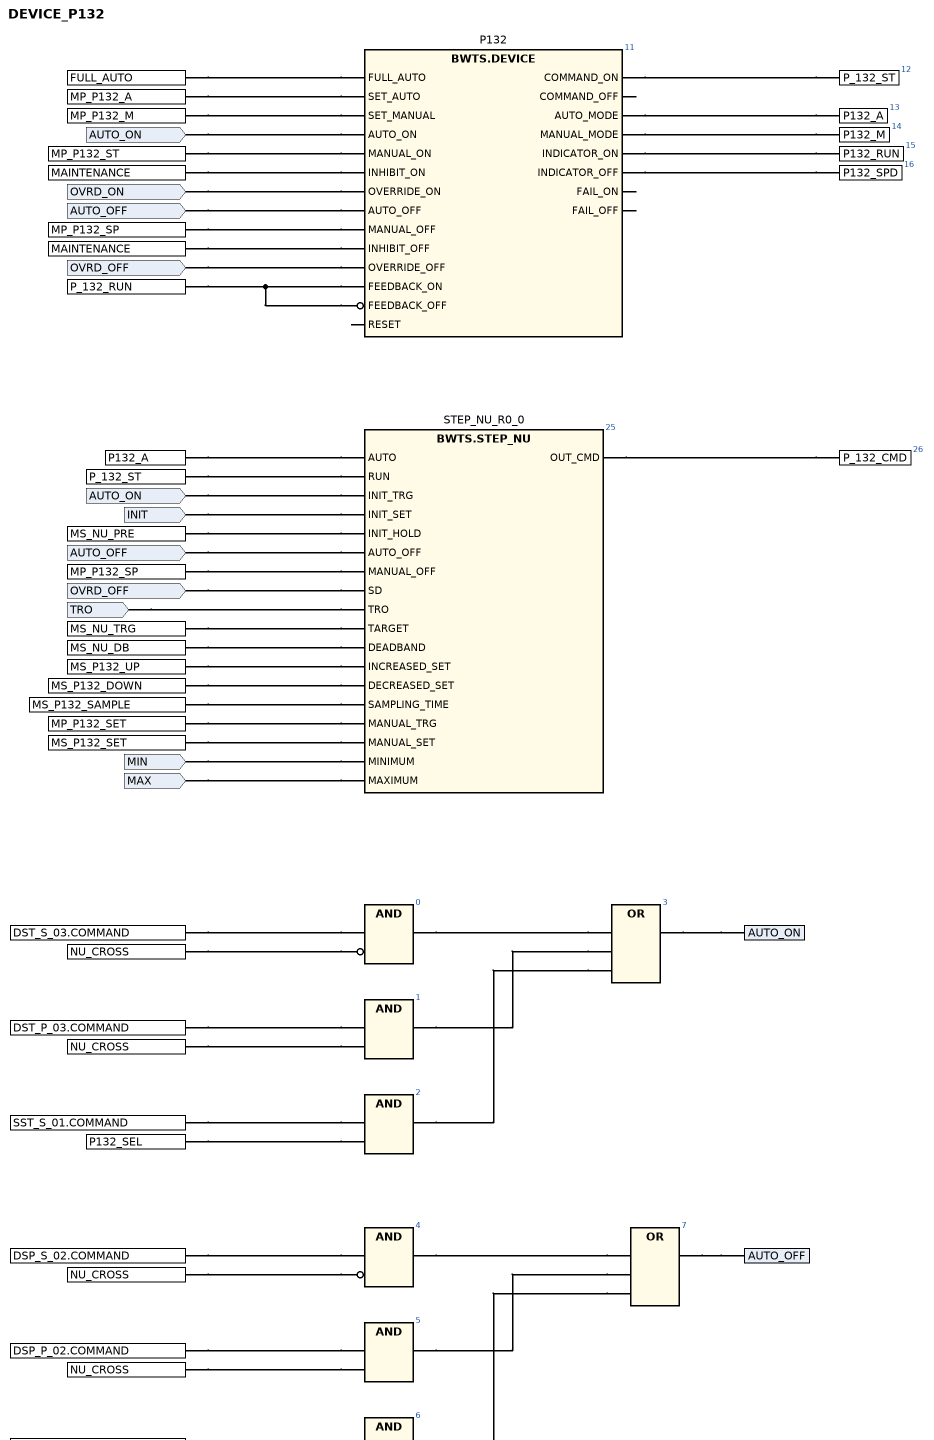
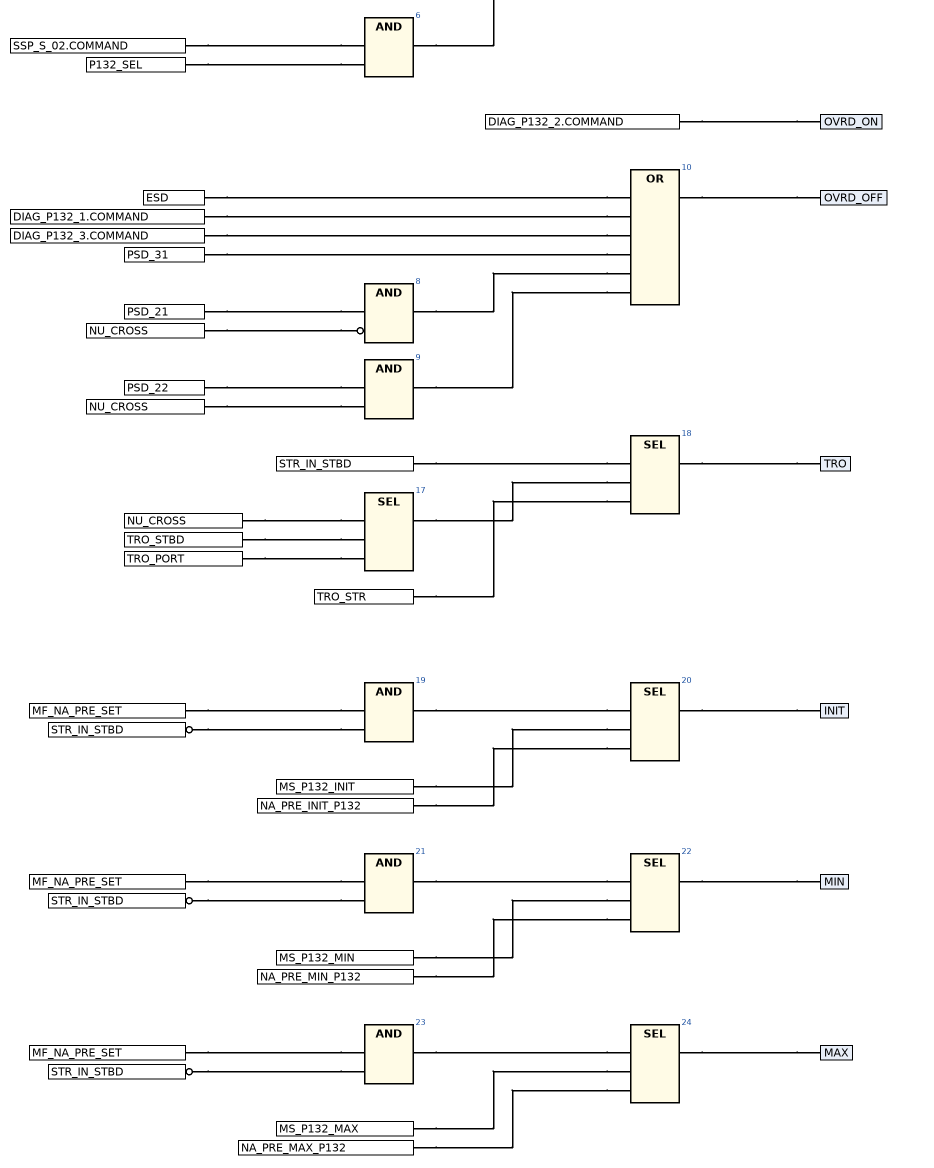
(* DST_S_03.COMMAND AND NOT NU_CROSS OR DST_P_03.COMMAND AND NU_CROSS OR SST_S_01.COMMAND AND P132_SEL; result not used *)
(* DSP_S_02.COMMAND AND NOT NU_CROSS OR DSP_P_02.COMMAND AND NU_CROSS OR SSP_S_02.COMMAND AND P132_SEL; result not used *)
(* ESD OR DIAG_P132_1.COMMAND OR DIAG_P132_3.COMMAND OR PSD_31 OR PSD_21 AND NOT NU_CROSS OR PSD_22 AND NU_CROSS; result not used *)
P132(
    FULL_AUTO := FULL_AUTO,
    SET_AUTO := MP_P132_A,
    SET_MANUAL := MP_P132_M,
    AUTO_ON := _w1,
    MANUAL_ON := MP_P132_ST,
    INHIBIT_ON := MAINTENANCE,
    OVERRIDE_ON := _w2,
    AUTO_OFF := _w3,
    MANUAL_OFF := MP_P132_SP,
    INHIBIT_OFF := MAINTENANCE,
    OVERRIDE_OFF := _w4,
    FEEDBACK_ON := P_132_RUN,
    FEEDBACK_OFF := NOT P_132_RUN); // BWTS.DEVICE
P_132_ST := P132.COMMAND_ON;
P132_A := P132.AUTO_MODE;
P132_M := P132.MANUAL_MODE;
P132_RUN := P132.INDICATOR_ON;
P132_SPD := P132.INDICATOR_OFF;
(* SEL(STR_IN_STBD, SEL(NU_CROSS, TRO_STBD, TRO_PORT), TRO_STR); result not used *)
(* SEL(MF_NA_PRE_SET AND NOT STR_IN_STBD, MS_P132_INIT, NA_PRE_INIT_P132); result not used *)
(* SEL(MF_NA_PRE_SET AND NOT STR_IN_STBD, MS_P132_MIN, NA_PRE_MIN_P132); result not used *)
(* SEL(MF_NA_PRE_SET AND NOT STR_IN_STBD, MS_P132_MAX, NA_PRE_MAX_P132); result not used *)
STEP_NU_R0_0(
    AUTO := P132_A,
    RUN := P_132_ST,
    INIT_TRG := _w5,
    INIT_SET := _w6,
    INIT_HOLD := MS_NU_PRE,
    AUTO_OFF := _w7,
    MANUAL_OFF := MP_P132_SP,
    SD := _w8,
    TRO := _w9,
    TARGET := MS_NU_TRG,
    DEADBAND := MS_NU_DB,
    INCREASED_SET := MS_P132_UP,
    DECREASED_SET := MS_P132_DOWN,
    SAMPLING_TIME := MS_P132_SAMPLE,
    MANUAL_TRG := MP_P132_SET,
    MANUAL_SET := MS_P132_SET,
    MINIMUM := _w10,
    MAXIMUM := _w11); // BWTS.STEP_NU
P_132_CMD := STEP_NU_R0_0.OUT_CMD;

END_PROGRAM

// Device/Application/Logic/4.Device/DEVICE_P232
PROGRAM DEVICE_P232
VAR
	P232 : BWTS.DEVICE;
	STEP_NU_R0_0: BWTS.STEP_NU;                                                                                                                            	
END_VAR
VAR // added by the converter: edge detectors and wires of the graphical bodies
    _w1, _w2, _w3, _w4, _w5, _w6, _w7, _w8, _w9, _w10, _w11 : ANY;
END_VAR

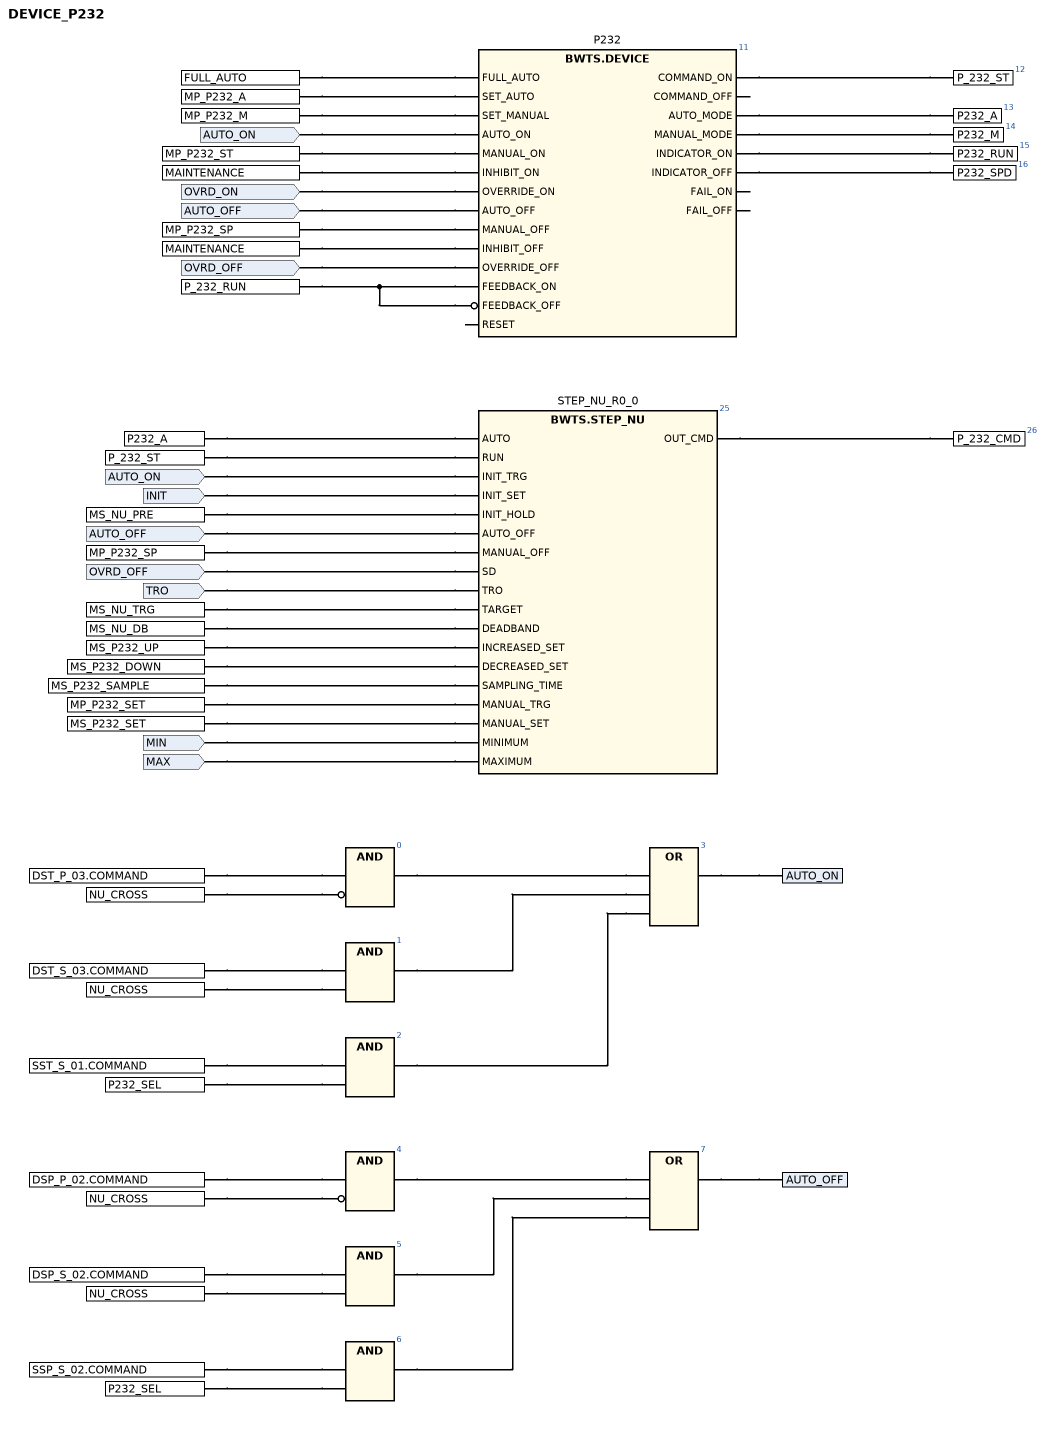
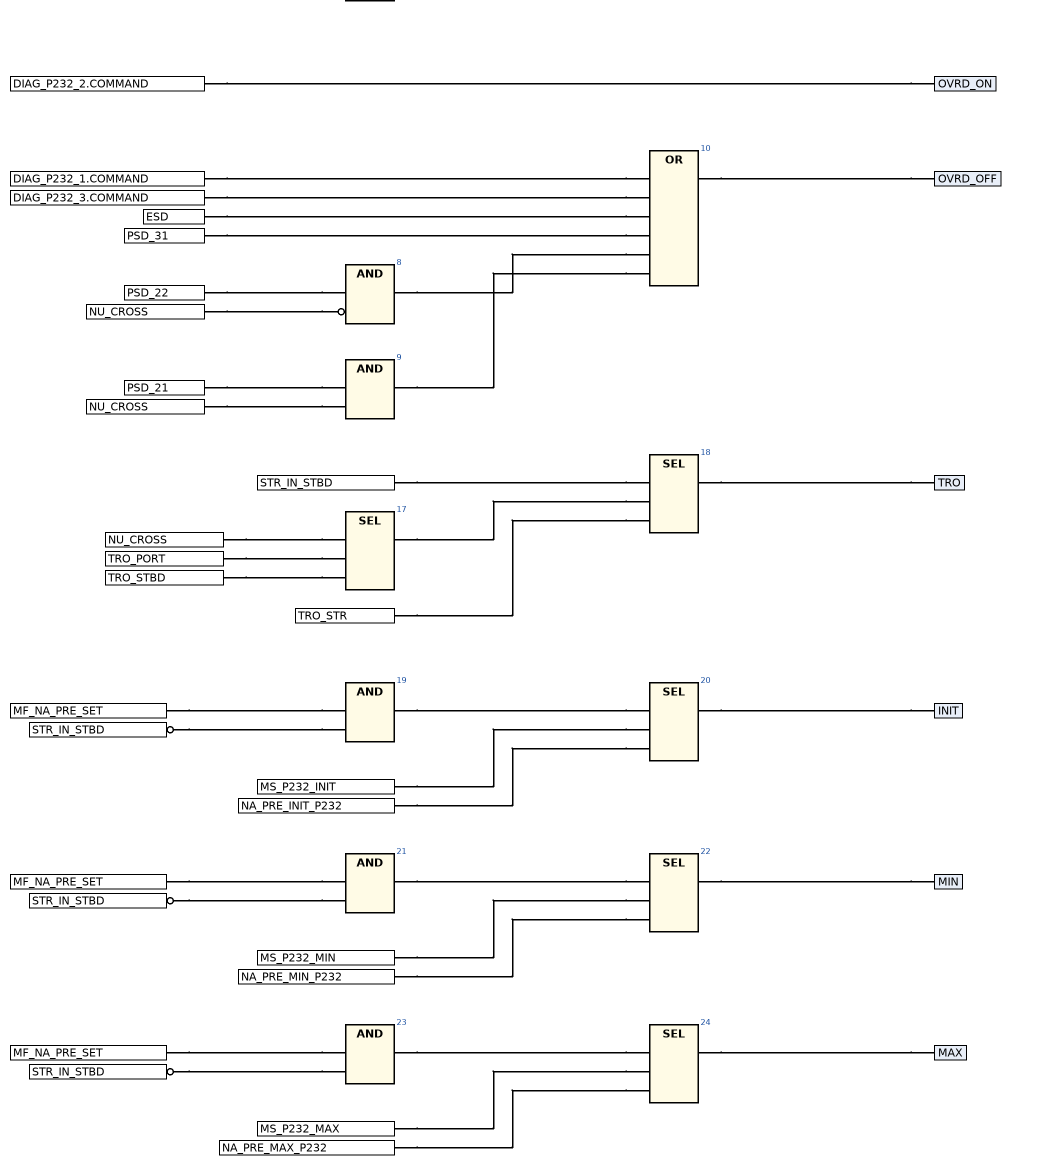
(* DST_P_03.COMMAND AND NOT NU_CROSS OR DST_S_03.COMMAND AND NU_CROSS OR SST_S_01.COMMAND AND P232_SEL; result not used *)
(* DSP_P_02.COMMAND AND NOT NU_CROSS OR DSP_S_02.COMMAND AND NU_CROSS OR SSP_S_02.COMMAND AND P232_SEL; result not used *)
(* DIAG_P232_1.COMMAND OR DIAG_P232_3.COMMAND OR ESD OR PSD_31 OR PSD_22 AND NOT NU_CROSS OR PSD_21 AND NU_CROSS; result not used *)
P232(
    FULL_AUTO := FULL_AUTO,
    SET_AUTO := MP_P232_A,
    SET_MANUAL := MP_P232_M,
    AUTO_ON := _w1,
    MANUAL_ON := MP_P232_ST,
    INHIBIT_ON := MAINTENANCE,
    OVERRIDE_ON := _w2,
    AUTO_OFF := _w3,
    MANUAL_OFF := MP_P232_SP,
    INHIBIT_OFF := MAINTENANCE,
    OVERRIDE_OFF := _w4,
    FEEDBACK_ON := P_232_RUN,
    FEEDBACK_OFF := NOT P_232_RUN); // BWTS.DEVICE
P_232_ST := P232.COMMAND_ON;
P232_A := P232.AUTO_MODE;
P232_M := P232.MANUAL_MODE;
P232_RUN := P232.INDICATOR_ON;
P232_SPD := P232.INDICATOR_OFF;
(* SEL(STR_IN_STBD, SEL(NU_CROSS, TRO_PORT, TRO_STBD), TRO_STR); result not used *)
(* SEL(MF_NA_PRE_SET AND NOT STR_IN_STBD, MS_P232_INIT, NA_PRE_INIT_P232); result not used *)
(* SEL(MF_NA_PRE_SET AND NOT STR_IN_STBD, MS_P232_MIN, NA_PRE_MIN_P232); result not used *)
(* SEL(MF_NA_PRE_SET AND NOT STR_IN_STBD, MS_P232_MAX, NA_PRE_MAX_P232); result not used *)
STEP_NU_R0_0(
    AUTO := P232_A,
    RUN := P_232_ST,
    INIT_TRG := _w5,
    INIT_SET := _w6,
    INIT_HOLD := MS_NU_PRE,
    AUTO_OFF := _w7,
    MANUAL_OFF := MP_P232_SP,
    SD := _w8,
    TRO := _w9,
    TARGET := MS_NU_TRG,
    DEADBAND := MS_NU_DB,
    INCREASED_SET := MS_P232_UP,
    DECREASED_SET := MS_P232_DOWN,
    SAMPLING_TIME := MS_P232_SAMPLE,
    MANUAL_TRG := MP_P232_SET,
    MANUAL_SET := MS_P232_SET,
    MINIMUM := _w10,
    MAXIMUM := _w11); // BWTS.STEP_NU
P_232_CMD := STEP_NU_R0_0.OUT_CMD;

END_PROGRAM

// Device/Application/Logic/4.Device/DEVICE_XV1171A
PROGRAM DEVICE_XV1171A
VAR
	XV1171A : BWTS.DEVICE;
END_VAR
VAR // added by the converter: edge detectors and wires of the graphical bodies
    _w1, _w2, _w3, _w4 : ANY;
END_VAR

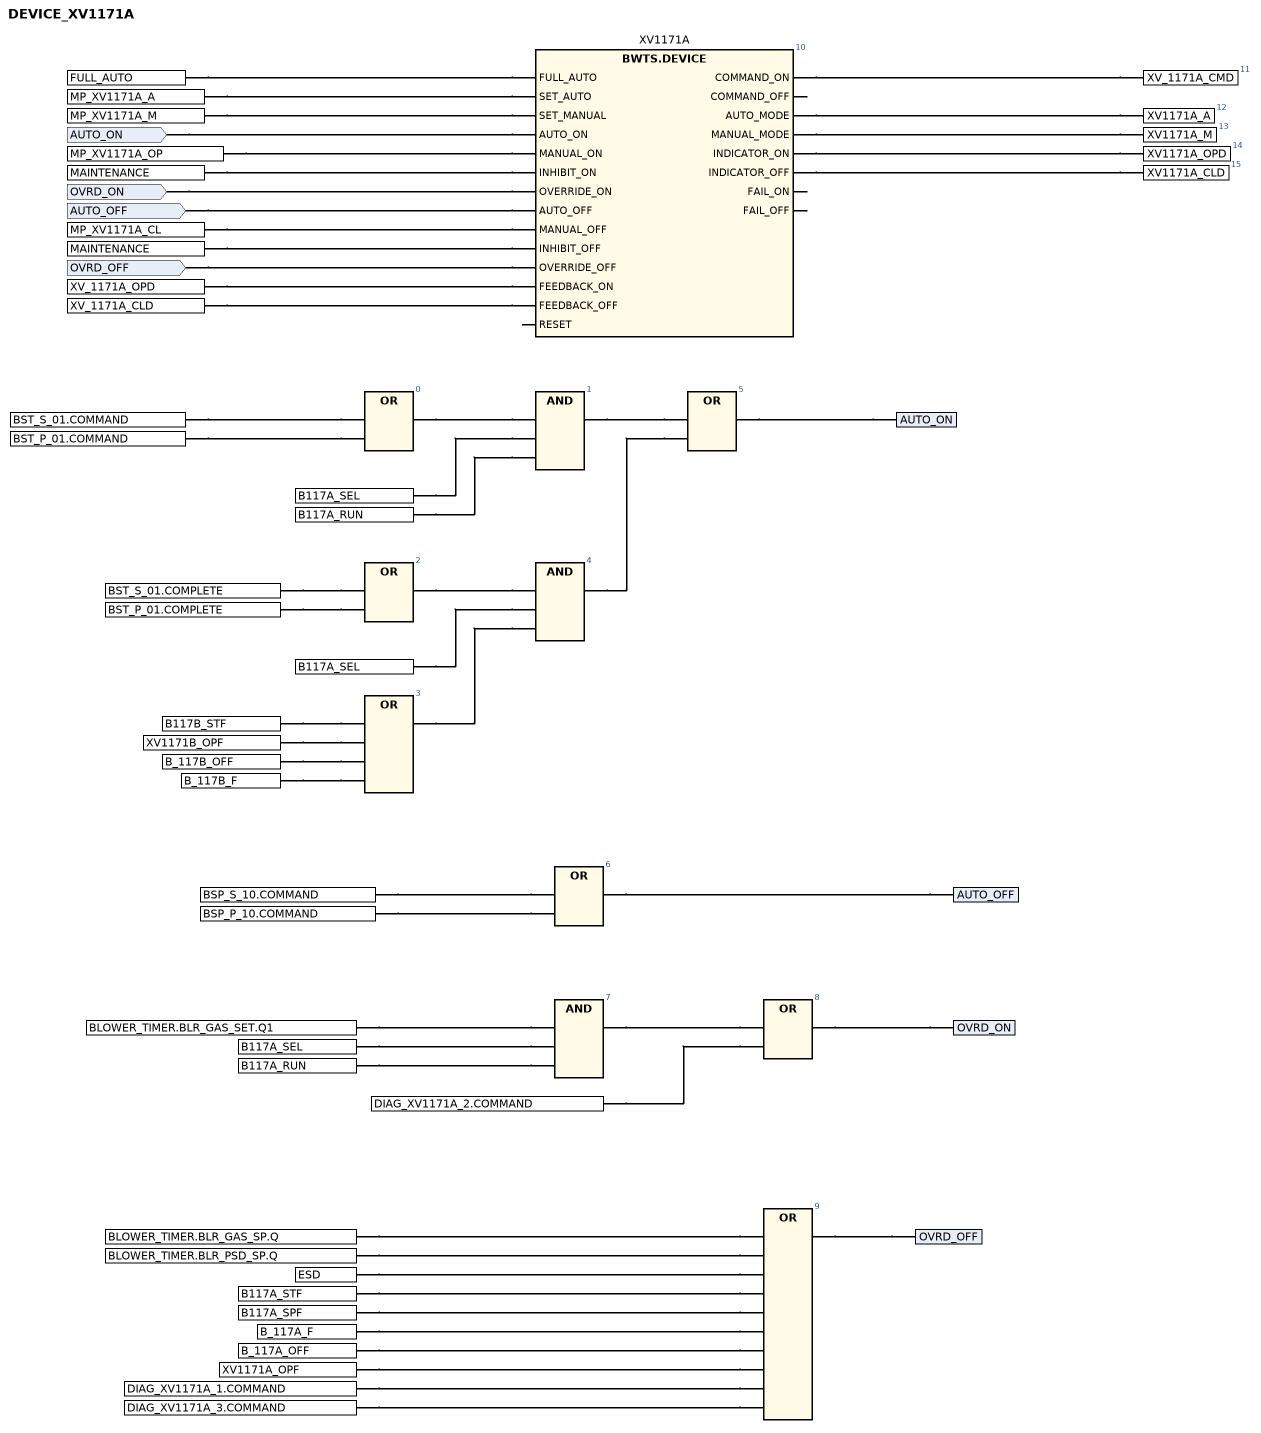
(* (BST_S_01.COMMAND OR BST_P_01.COMMAND) AND B117A_SEL AND B117A_RUN OR (BST_S_01.COMPLETE OR BST_P_01.COMPLETE) AND B117A_SEL AND (B117B_STF OR XV1171B_OPF OR B_117B_OFF OR B_117B_F); result not used *)
(* BSP_S_10.COMMAND OR BSP_P_10.COMMAND; result not used *)
(* BLOWER_TIMER.BLR_GAS_SET.Q1 AND B117A_SEL AND B117A_RUN OR DIAG_XV1171A_2.COMMAND; result not used *)
(* BLOWER_TIMER.BLR_GAS_SP.Q OR BLOWER_TIMER.BLR_PSD_SP.Q OR ESD OR B117A_STF OR B117A_SPF OR B_117A_F OR B_117A_OFF OR XV1171A_OPF OR DIAG_XV1171A_1.COMMAND OR DIAG_XV1171A_3.COMMAND; result not used *)
XV1171A(
    FULL_AUTO := FULL_AUTO,
    SET_AUTO := MP_XV1171A_A,
    SET_MANUAL := MP_XV1171A_M,
    AUTO_ON := _w1,
    MANUAL_ON := MP_XV1171A_OP,
    INHIBIT_ON := MAINTENANCE,
    OVERRIDE_ON := _w2,
    AUTO_OFF := _w3,
    MANUAL_OFF := MP_XV1171A_CL,
    INHIBIT_OFF := MAINTENANCE,
    OVERRIDE_OFF := _w4,
    FEEDBACK_ON := XV_1171A_OPD,
    FEEDBACK_OFF := XV_1171A_CLD); // BWTS.DEVICE
XV_1171A_CMD := XV1171A.COMMAND_ON;
XV1171A_A := XV1171A.AUTO_MODE;
XV1171A_M := XV1171A.MANUAL_MODE;
XV1171A_OPD := XV1171A.INDICATOR_ON;
XV1171A_CLD := XV1171A.INDICATOR_OFF;

END_PROGRAM

// Device/Application/Logic/4.Device/DEVICE_XV1171B
PROGRAM DEVICE_XV1171B
VAR
	XV1171B : BWTS.DEVICE;
END_VAR
VAR // added by the converter: edge detectors and wires of the graphical bodies
    _w1, _w2, _w3, _w4 : ANY;
END_VAR

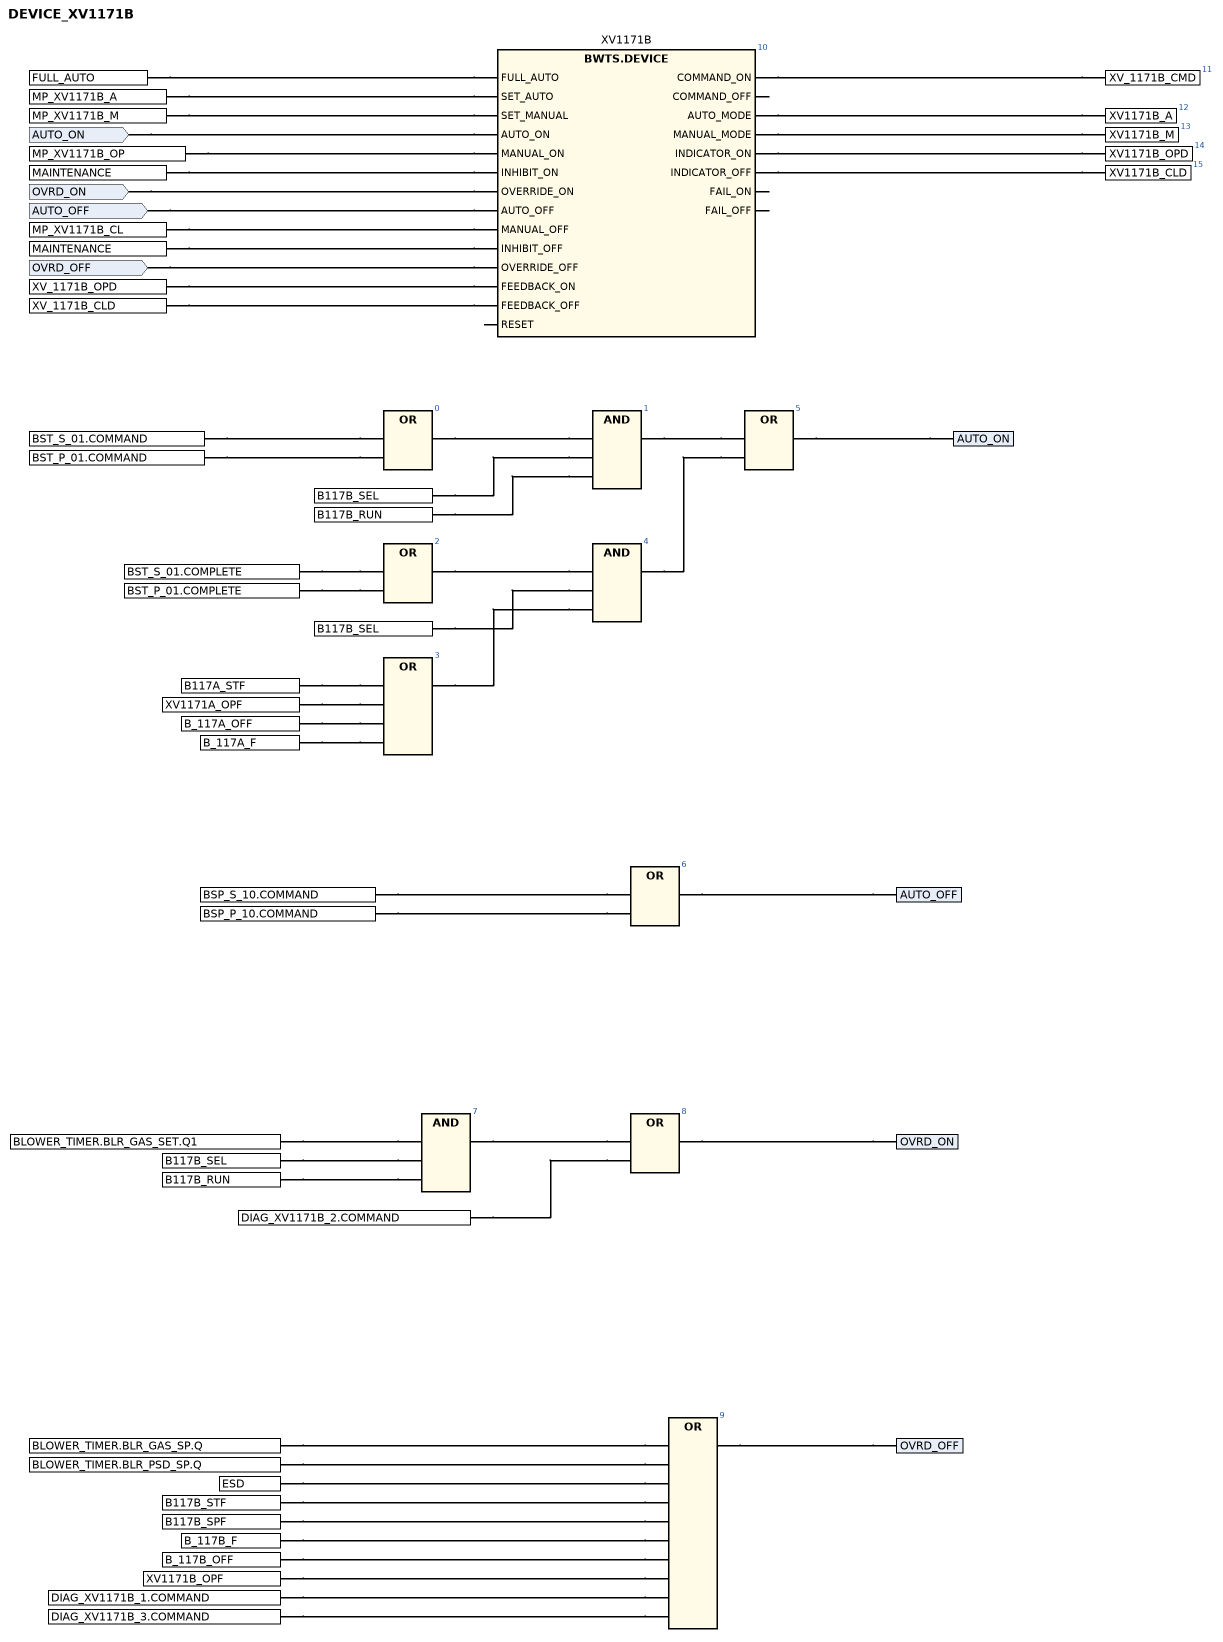
(* (BST_S_01.COMMAND OR BST_P_01.COMMAND) AND B117B_SEL AND B117B_RUN OR (BST_S_01.COMPLETE OR BST_P_01.COMPLETE) AND B117B_SEL AND (B117A_STF OR XV1171A_OPF OR B_117A_OFF OR B_117A_F); result not used *)
(* BSP_S_10.COMMAND OR BSP_P_10.COMMAND; result not used *)
(* BLOWER_TIMER.BLR_GAS_SET.Q1 AND B117B_SEL AND B117B_RUN OR DIAG_XV1171B_2.COMMAND; result not used *)
(* BLOWER_TIMER.BLR_GAS_SP.Q OR BLOWER_TIMER.BLR_PSD_SP.Q OR ESD OR B117B_STF OR B117B_SPF OR B_117B_F OR B_117B_OFF OR XV1171B_OPF OR DIAG_XV1171B_1.COMMAND OR DIAG_XV1171B_3.COMMAND; result not used *)
XV1171B(
    FULL_AUTO := FULL_AUTO,
    SET_AUTO := MP_XV1171B_A,
    SET_MANUAL := MP_XV1171B_M,
    AUTO_ON := _w1,
    MANUAL_ON := MP_XV1171B_OP,
    INHIBIT_ON := MAINTENANCE,
    OVERRIDE_ON := _w2,
    AUTO_OFF := _w3,
    MANUAL_OFF := MP_XV1171B_CL,
    INHIBIT_OFF := MAINTENANCE,
    OVERRIDE_OFF := _w4,
    FEEDBACK_ON := XV_1171B_OPD,
    FEEDBACK_OFF := XV_1171B_CLD); // BWTS.DEVICE
XV_1171B_CMD := XV1171B.COMMAND_ON;
XV1171B_A := XV1171B.AUTO_MODE;
XV1171B_M := XV1171B.MANUAL_MODE;
XV1171B_OPD := XV1171B.INDICATOR_ON;
XV1171B_CLD := XV1171B.INDICATOR_OFF;

END_PROGRAM

// Device/Application/Logic/4.Device/DEVICE_FCV1131
PROGRAM DEVICE_FCV1131
VAR
	FCV1131: BWTS.PID_CONT;

END_VAR
VAR // added by the converter: edge detectors and wires of the graphical bodies
    _w1, _w2, _w3, _w4, _w5, _w6, _w7 : ANY;
END_VAR

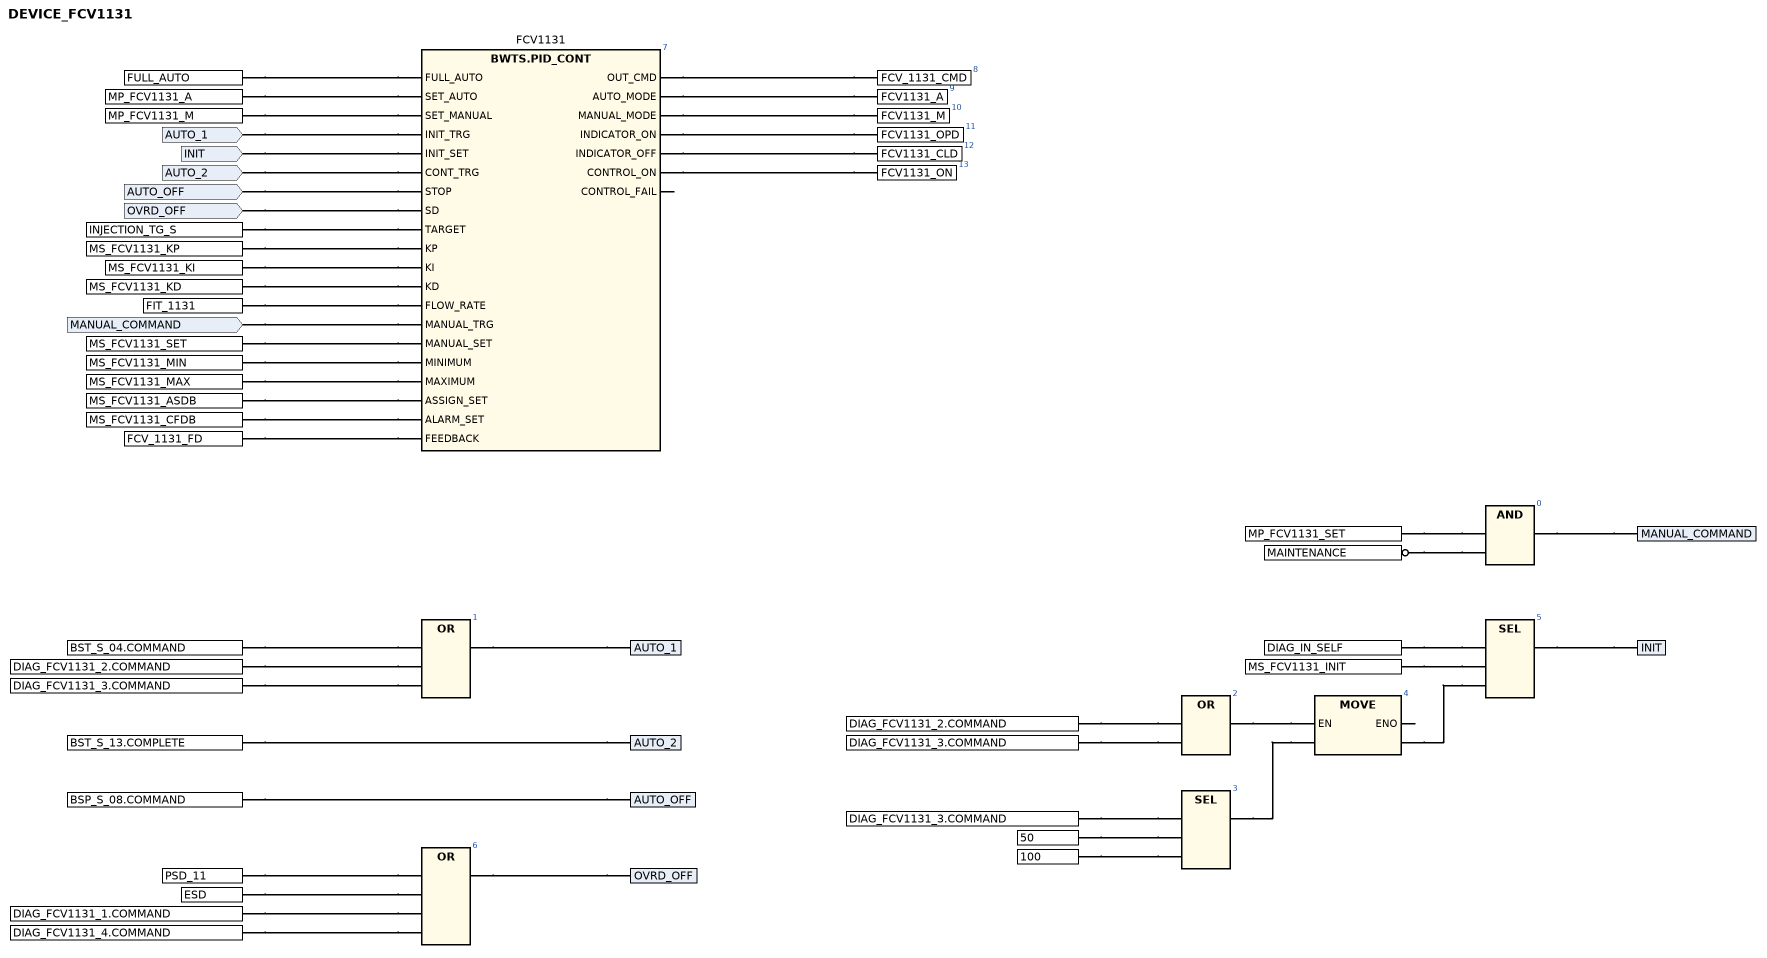
(* MP_FCV1131_SET AND NOT MAINTENANCE; result not used *)
(* BST_S_04.COMMAND OR DIAG_FCV1131_2.COMMAND OR DIAG_FCV1131_3.COMMAND; result not used *)
IF DIAG_FCV1131_2.COMMAND OR DIAG_FCV1131_3.COMMAND THEN _w1 := SEL(DIAG_FCV1131_3.COMMAND, 50, 100); END_IF
(* SEL(DIAG_IN_SELF, MS_FCV1131_INIT, _w1); result not used *)
(* PSD_11 OR ESD OR DIAG_FCV1131_1.COMMAND OR DIAG_FCV1131_4.COMMAND; result not used *)
FCV1131(
    FULL_AUTO := FULL_AUTO,
    SET_AUTO := MP_FCV1131_A,
    SET_MANUAL := MP_FCV1131_M,
    INIT_TRG := _w2,
    INIT_SET := _w3,
    CONT_TRG := _w4,
    STOP := _w5,
    SD := _w6,
    TARGET := INJECTION_TG_S,
    KP := MS_FCV1131_KP,
    KI := MS_FCV1131_KI,
    KD := MS_FCV1131_KD,
    FLOW_RATE := FIT_1131,
    MANUAL_TRG := _w7,
    MANUAL_SET := MS_FCV1131_SET,
    MINIMUM := MS_FCV1131_MIN,
    MAXIMUM := MS_FCV1131_MAX,
    ASSIGN_SET := MS_FCV1131_ASDB,
    ALARM_SET := MS_FCV1131_CFDB,
    FEEDBACK := FCV_1131_FD); // BWTS.PID_CONT
FCV_1131_CMD := FCV1131.OUT_CMD;
FCV1131_A := FCV1131.AUTO_MODE;
FCV1131_M := FCV1131.MANUAL_MODE;
FCV1131_OPD := FCV1131.INDICATOR_ON;
FCV1131_CLD := FCV1131.INDICATOR_OFF;
FCV1131_ON := FCV1131.CONTROL_ON;

END_PROGRAM

// Device/Application/Logic/4.Device/DEVICE_FCV2131
PROGRAM DEVICE_FCV2131
VAR
	FCV2131: BWTS.PID_CONT;

END_VAR
VAR // added by the converter: edge detectors and wires of the graphical bodies
    _w1, _w2, _w3, _w4, _w5, _w6, _w7 : ANY;
END_VAR

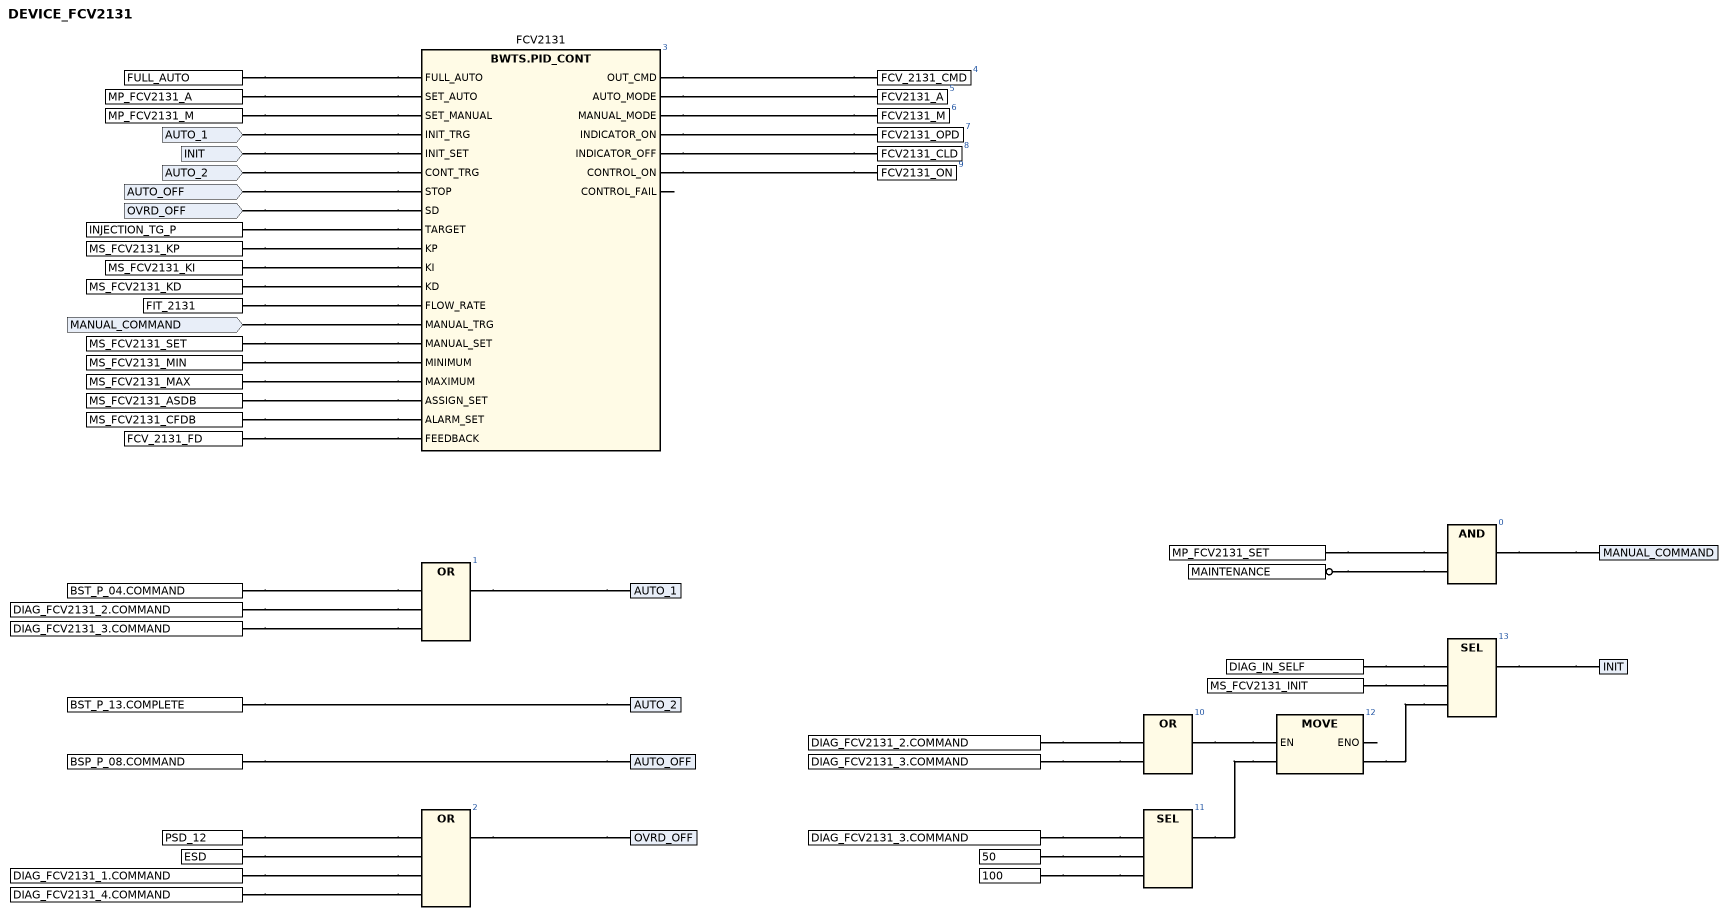
(* MP_FCV2131_SET AND NOT MAINTENANCE; result not used *)
(* BST_P_04.COMMAND OR DIAG_FCV2131_2.COMMAND OR DIAG_FCV2131_3.COMMAND; result not used *)
(* PSD_12 OR ESD OR DIAG_FCV2131_1.COMMAND OR DIAG_FCV2131_4.COMMAND; result not used *)
FCV2131(
    FULL_AUTO := FULL_AUTO,
    SET_AUTO := MP_FCV2131_A,
    SET_MANUAL := MP_FCV2131_M,
    INIT_TRG := _w1,
    INIT_SET := _w2,
    CONT_TRG := _w3,
    STOP := _w4,
    SD := _w5,
    TARGET := INJECTION_TG_P,
    KP := MS_FCV2131_KP,
    KI := MS_FCV2131_KI,
    KD := MS_FCV2131_KD,
    FLOW_RATE := FIT_2131,
    MANUAL_TRG := _w6,
    MANUAL_SET := MS_FCV2131_SET,
    MINIMUM := MS_FCV2131_MIN,
    MAXIMUM := MS_FCV2131_MAX,
    ASSIGN_SET := MS_FCV2131_ASDB,
    ALARM_SET := MS_FCV2131_CFDB,
    FEEDBACK := FCV_2131_FD); // BWTS.PID_CONT
FCV_2131_CMD := FCV2131.OUT_CMD;
FCV2131_A := FCV2131.AUTO_MODE;
FCV2131_M := FCV2131.MANUAL_MODE;
FCV2131_OPD := FCV2131.INDICATOR_ON;
FCV2131_CLD := FCV2131.INDICATOR_OFF;
FCV2131_ON := FCV2131.CONTROL_ON;
IF DIAG_FCV2131_2.COMMAND OR DIAG_FCV2131_3.COMMAND THEN _w7 := SEL(DIAG_FCV2131_3.COMMAND, 50, 100); END_IF
(* SEL(DIAG_IN_SELF, MS_FCV2131_INIT, _w7); result not used *)

END_PROGRAM

// Device/Application/Logic/4.Device/DEVICE_FCV1211
PROGRAM DEVICE_FCV1211
VAR
	INIT_SET : REAL;
	FCV1211: BWTS.STEP_FCV;
END_VAR
VAR // added by the converter: edge detectors and wires of the graphical bodies
    _w1, _w2, _w3, _w4, _w5, _w6, _w7, _w8, _w9 : ANY;
END_VAR

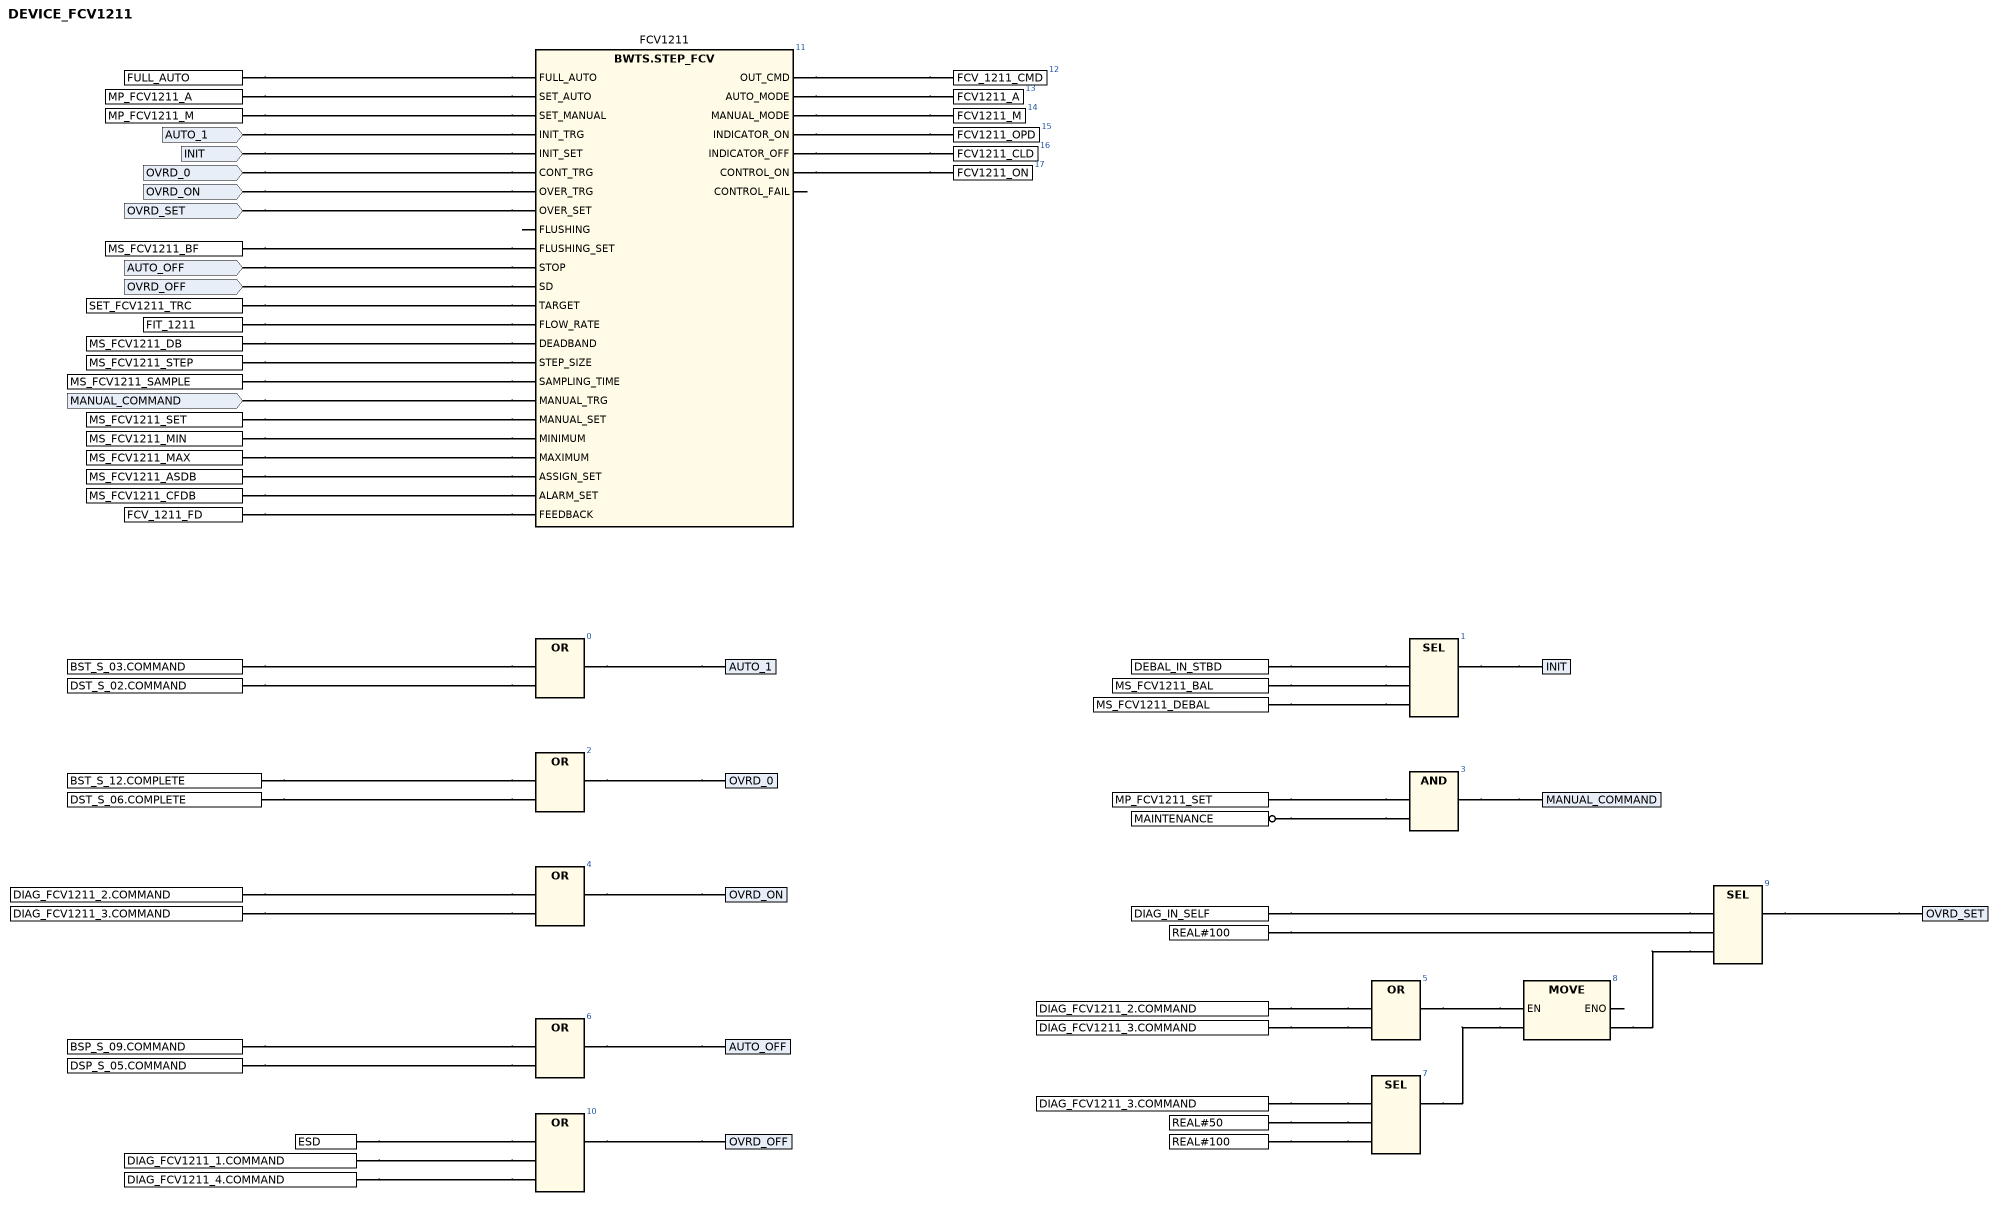
(* BST_S_03.COMMAND OR DST_S_02.COMMAND; result not used *)
(* SEL(DEBAL_IN_STBD, MS_FCV1211_BAL, MS_FCV1211_DEBAL); result not used *)
(* BST_S_12.COMPLETE OR DST_S_06.COMPLETE; result not used *)
(* MP_FCV1211_SET AND NOT MAINTENANCE; result not used *)
(* DIAG_FCV1211_2.COMMAND OR DIAG_FCV1211_3.COMMAND; result not used *)
(* BSP_S_09.COMMAND OR DSP_S_05.COMMAND; result not used *)
IF DIAG_FCV1211_2.COMMAND OR DIAG_FCV1211_3.COMMAND THEN _w1 := SEL(DIAG_FCV1211_3.COMMAND, REAL#50, REAL#100); END_IF
(* SEL(DIAG_IN_SELF, REAL#100, _w1); result not used *)
(* ESD OR DIAG_FCV1211_1.COMMAND OR DIAG_FCV1211_4.COMMAND; result not used *)
FCV1211(
    FULL_AUTO := FULL_AUTO,
    SET_AUTO := MP_FCV1211_A,
    SET_MANUAL := MP_FCV1211_M,
    INIT_TRG := _w2,
    INIT_SET := _w3,
    CONT_TRG := _w4,
    OVER_TRG := _w5,
    OVER_SET := _w6,
    FLUSHING_SET := MS_FCV1211_BF,
    STOP := _w7,
    SD := _w8,
    TARGET := SET_FCV1211_TRC,
    FLOW_RATE := FIT_1211,
    DEADBAND := MS_FCV1211_DB,
    STEP_SIZE := MS_FCV1211_STEP,
    SAMPLING_TIME := MS_FCV1211_SAMPLE,
    MANUAL_TRG := _w9,
    MANUAL_SET := MS_FCV1211_SET,
    MINIMUM := MS_FCV1211_MIN,
    MAXIMUM := MS_FCV1211_MAX,
    ASSIGN_SET := MS_FCV1211_ASDB,
    ALARM_SET := MS_FCV1211_CFDB,
    FEEDBACK := FCV_1211_FD); // BWTS.STEP_FCV
FCV_1211_CMD := FCV1211.OUT_CMD;
FCV1211_A := FCV1211.AUTO_MODE;
FCV1211_M := FCV1211.MANUAL_MODE;
FCV1211_OPD := FCV1211.INDICATOR_ON;
FCV1211_CLD := FCV1211.INDICATOR_OFF;
FCV1211_ON := FCV1211.CONTROL_ON;

END_PROGRAM

// Device/Application/Logic/4.Device/DEVICE_FCV2211
 PROGRAM DEVICE_FCV2211
VAR
	INIT_SET : REAL;
	FCV2211: BWTS.STEP_FCV;
END_VAR
VAR // added by the converter: edge detectors and wires of the graphical bodies
    _w1, _w2, _w3, _w4, _w5, _w6, _w7, _w8, _w9 : ANY;
END_VAR

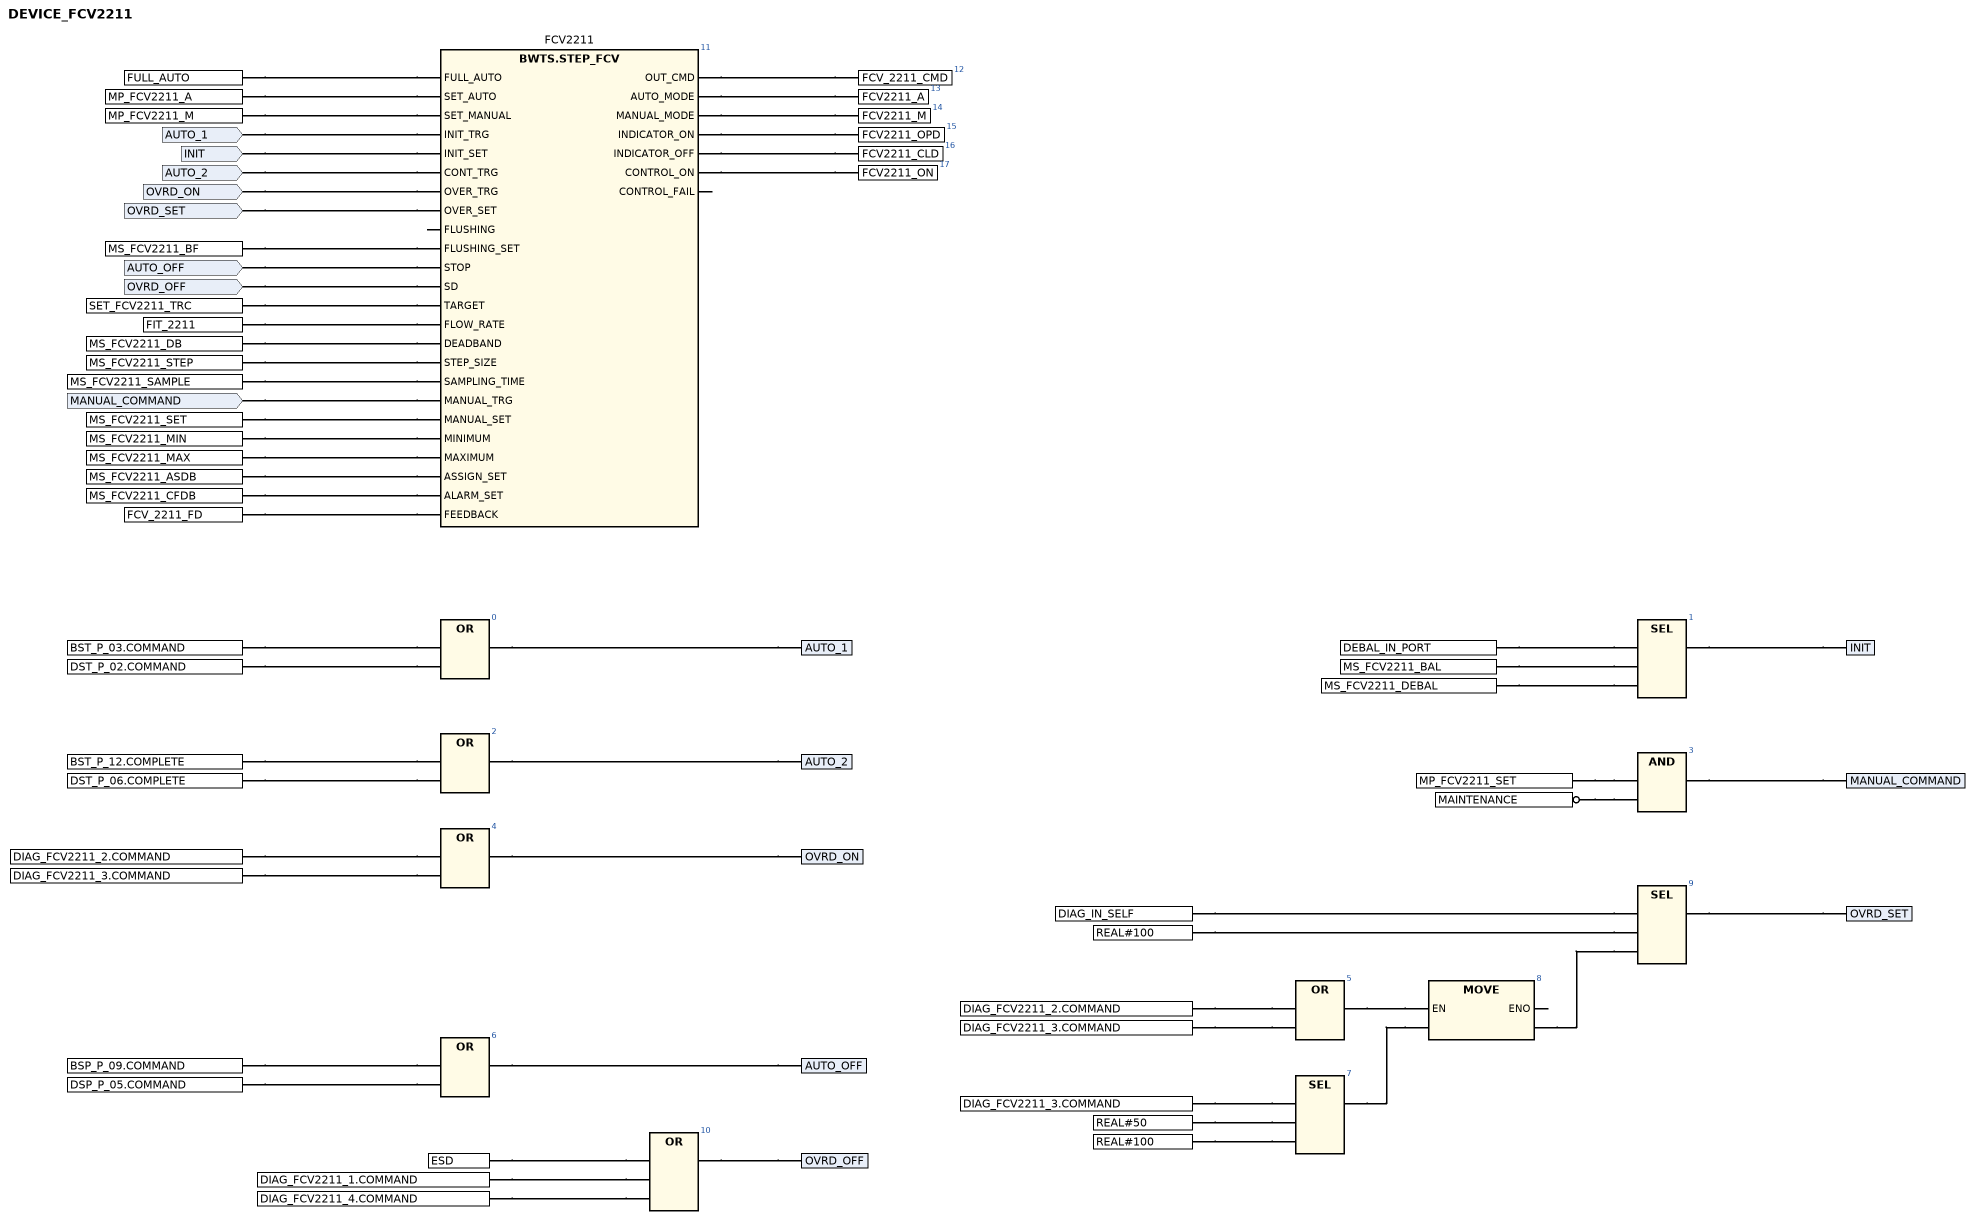
(* BST_P_03.COMMAND OR DST_P_02.COMMAND; result not used *)
(* SEL(DEBAL_IN_PORT, MS_FCV2211_BAL, MS_FCV2211_DEBAL); result not used *)
(* BST_P_12.COMPLETE OR DST_P_06.COMPLETE; result not used *)
(* MP_FCV2211_SET AND NOT MAINTENANCE; result not used *)
(* DIAG_FCV2211_2.COMMAND OR DIAG_FCV2211_3.COMMAND; result not used *)
(* BSP_P_09.COMMAND OR DSP_P_05.COMMAND; result not used *)
IF DIAG_FCV2211_2.COMMAND OR DIAG_FCV2211_3.COMMAND THEN _w1 := SEL(DIAG_FCV2211_3.COMMAND, REAL#50, REAL#100); END_IF
(* SEL(DIAG_IN_SELF, REAL#100, _w1); result not used *)
(* ESD OR DIAG_FCV2211_1.COMMAND OR DIAG_FCV2211_4.COMMAND; result not used *)
FCV2211(
    FULL_AUTO := FULL_AUTO,
    SET_AUTO := MP_FCV2211_A,
    SET_MANUAL := MP_FCV2211_M,
    INIT_TRG := _w2,
    INIT_SET := _w3,
    CONT_TRG := _w4,
    OVER_TRG := _w5,
    OVER_SET := _w6,
    FLUSHING_SET := MS_FCV2211_BF,
    STOP := _w7,
    SD := _w8,
    TARGET := SET_FCV2211_TRC,
    FLOW_RATE := FIT_2211,
    DEADBAND := MS_FCV2211_DB,
    STEP_SIZE := MS_FCV2211_STEP,
    SAMPLING_TIME := MS_FCV2211_SAMPLE,
    MANUAL_TRG := _w9,
    MANUAL_SET := MS_FCV2211_SET,
    MINIMUM := MS_FCV2211_MIN,
    MAXIMUM := MS_FCV2211_MAX,
    ASSIGN_SET := MS_FCV2211_ASDB,
    ALARM_SET := MS_FCV2211_CFDB,
    FEEDBACK := FCV_2211_FD); // BWTS.STEP_FCV
FCV_2211_CMD := FCV2211.OUT_CMD;
FCV2211_A := FCV2211.AUTO_MODE;
FCV2211_M := FCV2211.MANUAL_MODE;
FCV2211_OPD := FCV2211.INDICATOR_ON;
FCV2211_CLD := FCV2211.INDICATOR_OFF;
FCV2211_ON := FCV2211.CONTROL_ON;

END_PROGRAM

// Device/Application/Logic/0.ALARM/ALARM_INTERLOCK_A
PROGRAM ALARM_INTERLOCK_A
VAR

	ALARM_A_PT_1721,
	ALARM_A_PT_1722,
	ALARM_A_P_171,
	ALARM_A_PT_1121,
	ALARM_A_AIT_1121,
	ALARM_A_AIT_1122,
	ALARM_A_AIT_1123,
	ALARM_A_TE_1111,
	ALARM_A_CT_1111,	
	ALARM_A_FIT_1131,
	ALARM_A_FIT_2131,
	
	ALARM_A_FIT_1211,
	ALARM_A_FIT_2211,
	
	ALARM_A_LIT_1311,
	ALARM_A_AP_LVL_01
	: BWTS.ALARM_A;
END_VAR
VAR // added by the converter: edge detectors and wires of the graphical bodies
    _w1, _w2, _w3, _w4, _w5, _w6, _w7, _w8, _w9, _w10, _w11, _w12, _w13, _w14, _w15, _w16, _w17, _w18, _w19, _w20, _w21, _w22, _w23, _w24, _w25, _w26, _w27, _w28, _w29, _w30, _w31, _w32, _w33, _w34, _w35, _w36 : ANY;
END_VAR

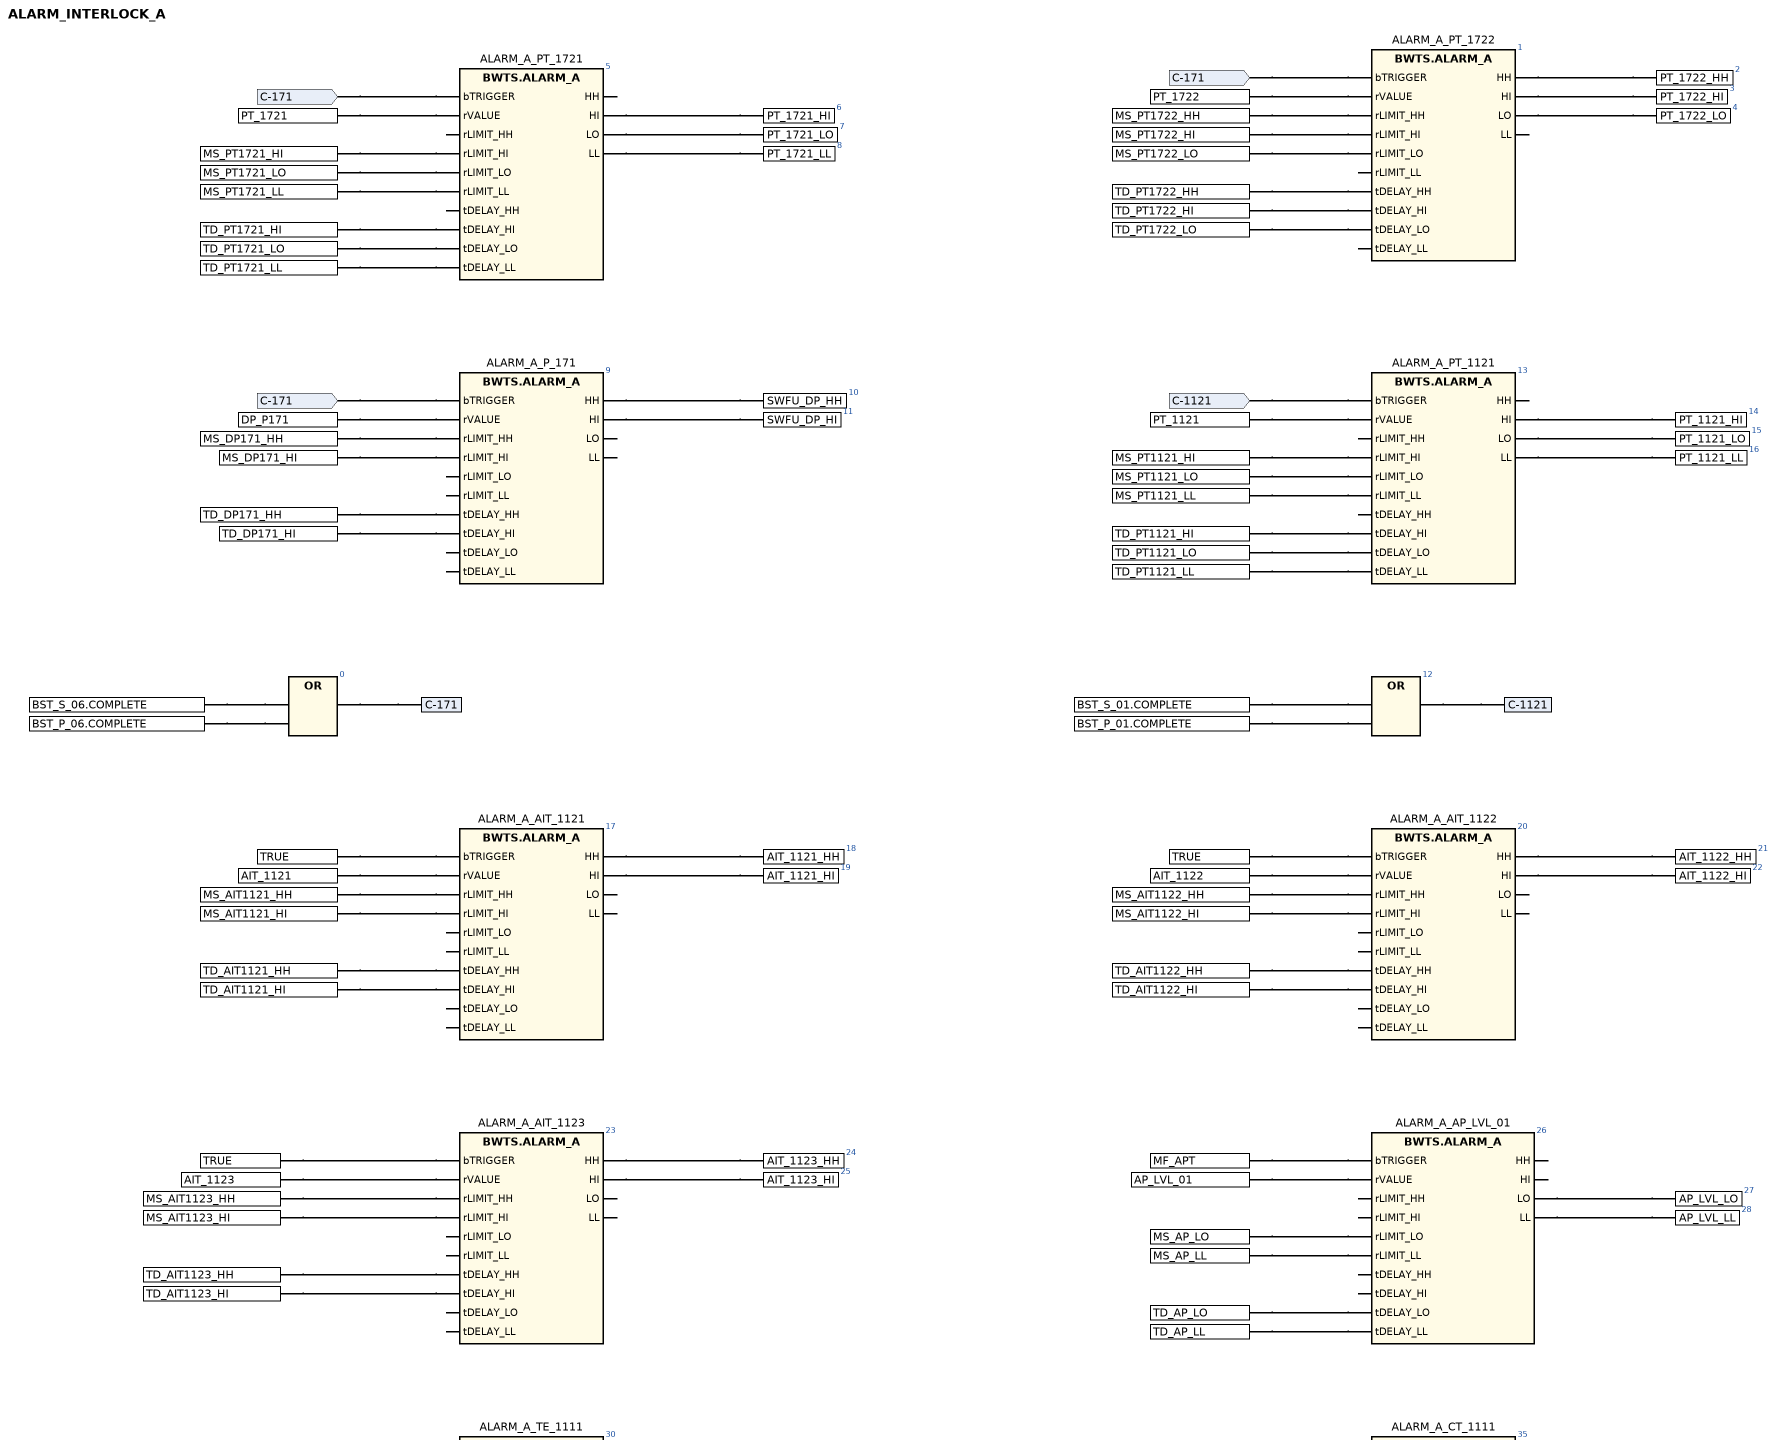
